(* Logix 5000 project; controller cal1615 1756-L62 rev 20.19; software revision 20.05; part 8 of 82 *)
(* tags used below, declared in another part *)
   AFI : BOOL;   // Always False Bit
   AutoT : PIDE_AUTOTUNE;
   FAULT : BOOL;   // Fault AFI
   HMI : BOOL;   // AFI HMI
   p01_dint_to_hmi : DINT[16];   // System Dint to HMI
   p01_param_heater_hl : REAL;   // Machine Parameter Heater HighTemperature Max Limit
   p01_param_process_air_hl : REAL;   // Machine Parameter Process Air High Limit
   p01_param_process_air_max : REAL;   // Machine Parameter Process Air High Temperature Max Setpoint Limit
   p01_param_temp_limit : REAL;   // Machine Parameter Maximum Temperature for Fan Operation
   p01_recipe_active : recipe;   // Active Recipe
   p01r01 : routine;
   p01r02 : routine;   // System Misc Control
   p01r02_all_fans_stopped : BOOL;   // System Misc Control All Fans Stopped
   p01r02_batch_run_time : DINT;   // System Misc Control Batch Minutes
   p01r02_batch_run_time_hrs : DINT;   // System Misc Control Batch Hours
   p01r02_ethernet_comm : DINT;
   p01r02_fault_exists : BOOL;
   p01r02_flash_bit : BOOL;   // System Misc Control Flash Bit
   p01r02_flash_timer_off : TIMER;   // System Misc Control Flash Timer Off
   p01r02_flash_timer_on : TIMER;   // System Misc Control Flash Timer On
   p01r02_plc_faults : DINT;   // System Misc Control PLC Faults
   p01r02_plc_scan_time : DINT;   // System PLC Scan Time
   p01r02_plc_scan_time_in_sec : REAL;   // System PLC Scan Time in Seconds
   p01r02_timer_batch : TIMER;   // System Misc Control Batch Timer Seconds
   p01r02_timer_fault : TIMER[25];   // System Misc Control Fault Dwell Timer
   p01r02_timer_half_second_off : TIMER;   // System Misc Control Timer Second Pulse Off
   p01r02_timer_half_second_on : TIMER;   // System Misc Control Timer 1/2 Second Pulse On
   p01r02_timer_second : TIMER[2];   // System Misc Control Timer Second Pulse
   p01r02_unack_fault : BOOL;   // System Misc Control Unacknowledged Fault Exists
   p01r02_unack_warning : BOOL;   // System Misc Control Unacknowledged Warning Exists
   p01r02_vfd_comm_2 : DINT[50];
   p01r02_warnings_exists : BOOL;
   p01r03 : routine;   // System Inputs
   p01r04 : routine;   // System Outputs
   p01r05 : routine;   // System Dint to HMI
   p01r06 : routine;   // System Real to HMI
   p01r07 : routine;   // System Alarms
   p01r08 : routine;   // System Warnings
   p01r09 : routine;   // System Modes
   p01r09_pb_global_reset : BOOL;   // System Modes PB: Global Fault Reset
   p01r10 : routine;   // System Annunciators
   p01r11 : routine;   // System Timer Presets
   p01r12 : routine;   // System Line Accel Decel Control
   p01r13 : routine;   // System Line Start Sequence
   p01r13_line_running : BOOL;   // System Line Start Sequence Line Running
   p02_dint_from_hmi : hmi_dint;
   p11r31_request_auto_run : BOOL;   // Zone 1 Exhaust Fan Run Request
   p11r32_request_auto_run : BOOL;   // Zone 1 Recirc Fan Run Request
   p12r31_request_auto_run : BOOL;   // Zone 2 Exhaust Fan Run Request
   p12r32_request_auto_run : BOOL;   // Zone 2 Recirc Fan Run Request
   p13r31_request_auto_run : BOOL;   // Zone 3 Exhaust Fan Run Request
   p13r32_request_auto_run : BOOL;   // Zone 3 Recirc Fan Run Request
   p23_do_enable_impreg_exhaust_fan : BOOL;   // Impreg Enclosure Digital Output Exhaust Fan Enable
   p23r13_request_auto_run : BOOL;   // Impreg Supply Fan VFD Request Auto Run
   p25_ai_ts2_lc : REAL;   // System Metering Roll VFD Minimum Start Tension
   p25r10_pid_manual_request : BOOL;
   p25r10_tension_request : BOOL;
   p25r20_pide_cv : REAL;

        [421] := 3.25, [422] := 3.25, [423] := 3.25, [424] := 3.25, [425] := 3.25, [426] := 3.25, [427] := 3.25, [428] := 3.25, [429] := 3.25, [430] := 3.25, [431] := 3.25, [432] := 3.25, [433] := 3.25, [434] := 3.25, [435] := 3.25, [436] := 3.25, [437] := 3.25, [438] := 3.25, [439] := 3.25, [440] := 3.25, [441] := 3.25, [442] := 3.25, [443] := 3.25, [444] := 3.25, [445] := 3.25, [446] := 3.25, [447] := 3.25, [448] := 3.25, [449] := 3.25, [450] := 3.25, [451] := 3.25, [452] := 3.25, [453] := 3.25, [454] := 3.25, [455] := 3.25, [456] := 3.25, [457] := 3.25, [458] := 3.25, [459] := 3.25, [460] := 3.25, [461] := 3.25, [462] := 3.25, [463] := 3.25, [464] := 3.25, [465] := 3.25, [466] := 3.25, [467] := 3.25, [468] := 3.25, [469] := 3.25, [470] := 3.25, [471] := 3.25, [472] := 3.25, [473] := 3.25, [474] := 3.25, [475] := 3.25, [476] := 3.25, [477] := 3.25, [478] := 3.25, [479] := 3.25, [480] := 3.25,
        [481] := 3.25, [482] := 3.25, [483] := 3.25, [484] := 3.25, [485] := 3.25, [486] := 3.25, [487] := 3.25, [488] := 3.25, [489] := 3.25, [490] := 3.25, [491] := 3.25, [492] := 3.25, [493] := 3.25, [494] := 3.25, [495] := 3.25, [496] := 3.25, [497] := 3.25, [498] := 3.25, [499] := 3.25, [500] := 3.25, [501] := 3.25, [502] := 3.25, [503] := 3.25, [504] := 3.25, [505] := 3.25, [506] := 3.25, [507] := 3.25, [508] := 3.25, [509] := 3.25, [510] := 3.25, [511] := 3.25, [512] := 3.25, [513] := 3.25, [514] := 3.25, [515] := 3.25, [516] := 3.25, [517] := 3.25, [518] := 3.25, [519] := 3.25, [520] := 3.25, [521] := 3.25, [522] := 3.25, [523] := 3.25, [524] := 3.25, [525] := 3.25, [526] := 3.25, [527] := 3.25, [528] := 3.25, [529] := 3.25, [530] := 3.25, [531] := 3.25, [532] := 3.25, [533] := 3.25, [534] := 3.25, [535] := 3.25, [536] := 3.25, [537] := 3.25, [538] := 3.25, [539] := 3.25, [540] := 3.25,
        [541] := 3.25, [542] := 3.25, [543] := 3.25, [544] := 3.25, [545] := 3.25, [546] := 3.25, [547] := 3.25, [548] := 3.25, [549] := 3.25, [550] := 3.25, [551] := 3.25, [552] := 3.25, [553] := 3.25, [554] := 3.25, [555] := 3.25, [556] := 3.25, [557] := 3.25, [558] := 3.25, [559] := 3.25, [560] := 3.25, [561] := 3.25, [562] := 3.25, [563] := 3.25, [564] := 3.25, [565] := 3.25, [566] := 3.25, [567] := 3.25, [568] := 3.25, [569] := 3.25, [570] := 3.25, [571] := 3.25, [572] := 3.25, [573] := 3.25, [574] := 3.25, [575] := 3.25, [576] := 3.25, [577] := 3.25, [578] := 3.25, [579] := 3.25, [580] := 3.25, [581] := 3.25, [582] := 3.25, [583] := 3.25, [584] := 3.25, [585] := 3.25, [586] := 3.25, [587] := 3.25, [588] := 3.25, [589] := 3.25, [590] := 3.25, [591] := 3.25, [592] := 3.25, [593] := 3.25, [594] := 3.25, [595] := 3.25, [596] := 3.25, [597] := 3.25, [598] := 3.25, [599] := 3.25, [600] := 3.25,
        [601] := 3.25, [602] := 3.25, [603] := 3.25, [604] := 3.25, [605] := 3.25, [606] := 3.25, [607] := 3.25, [608] := 3.25, [609] := 3.25, [610] := 3.25, [611] := 3.25, [612] := 3.25, [613] := 3.25, [614] := 3.25, [615] := 3.25, [616] := 3.25, [617] := 3.25, [618] := 3.25, [619] := 3.25, [620] := 3.25, [621] := 3.25, [622] := 3.25, [623] := 3.25, [624] := 3.25, [625] := 3.25, [626] := 3.25, [627] := 3.25, [628] := 3.25, [629] := 3.25, [630] := 3.25, [631] := 3.25, [632] := 3.25, [633] := 3.25, [634] := 3.25, [635] := 3.25, [636] := 3.25, [637] := 3.25, [638] := 3.25, [639] := 3.25, [640] := 3.25, [641] := 3.25, [642] := 3.25, [643] := 3.25, [644] := 3.25, [645] := 3.25, [646] := 3.25, [647] := 3.25, [648] := 3.25, [649] := 3.25, [650] := 3.25, [651] := 3.25, [652] := 3.25, [653] := 3.25, [654] := 3.25, [655] := 3.25, [656] := 3.25, [657] := 3.25, [658] := 3.25, [659] := 3.25, [660] := 3.25,
        [661] := 3.25, [662] := 3.25, [663] := 3.25, [664] := 3.25, [665] := 3.25, [666] := 3.25, [667] := 3.25, [668] := 3.25, [669] := 3.25, [670] := 3.25, [671] := 3.25, [672] := 3.25, [673] := 3.25, [674] := 3.25, [675] := 3.25, [676] := 3.25, [677] := 3.25, [678] := 3.25, [679] := 3.25, [680] := 3.25, [681] := 3.25, [682] := 3.25, [683] := 3.25, [684] := 3.25, [685] := 3.25, [686] := 3.25, [687] := 3.25, [688] := 3.25, [689] := 3.25, [690] := 3.25, [691] := 3.25, [692] := 3.25, [693] := 3.25, [694] := 3.25, [695] := 3.25, [696] := 3.25, [697] := 3.25, [698] := 3.25, [699] := 3.25, [700] := 3.25, [701] := 3.25, [702] := 3.25, [703] := 3.25, [704] := 3.25, [705] := 3.25, [706] := 3.25, [707] := 3.25, [708] := 3.25, [709] := 3.25, [710] := 3.25, [711] := 3.25, [712] := 3.25, [713] := 3.25, [714] := 3.25, [715] := 3.25, [716] := 3.25, [717] := 3.25, [718] := 3.25, [719] := 3.25, [720] := 3.25,
        [721] := 3.25, [722] := 3.25, [723] := 3.25, [724] := 3.25, [725] := 3.25, [726] := 3.25, [727] := 3.25, [728] := 3.25, [729] := 3.25, [730] := 3.25, [731] := 3.25, [732] := 3.25, [733] := 3.25, [734] := 3.25, [735] := 3.25, [736] := 3.25, [737] := 3.25, [738] := 3.25, [739] := 3.25, [740] := 3.25, [741] := 3.25, [742] := 3.25, [743] := 3.25, [744] := 3.25, [745] := 3.25, [746] := 3.25, [747] := 3.25, [748] := 3.25, [749] := 3.25, [750] := 3.25, [751] := 3.25, [752] := 3.25, [753] := 3.25, [754] := 3.25, [755] := 3.25, [756] := 3.25, [757] := 3.25, [758] := 3.25, [759] := 3.25, [760] := 3.25, [761] := 3.25, [762] := 3.25, [763] := 3.25, [764] := 3.25, [765] := 3.25, [766] := 3.25, [767] := 3.25, [768] := 3.25, [769] := 3.25, [770] := 3.25, [771] := 3.25, [772] := 3.25, [773] := 3.25, [774] := 3.25, [775] := 3.25, [776] := 3.25, [777] := 3.25, [778] := 3.25, [779] := 3.25, [780] := 3.25,
        [781] := 3.25, [782] := 3.25, [783] := 3.25, [784] := 3.25, [785] := 3.25, [786] := 3.25, [787] := 3.25, [788] := 3.25, [789] := 3.25, [790] := 3.25, [791] := 3.25, [792] := 3.25, [793] := 3.25, [794] := 3.25, [795] := 3.25, [796] := 3.25, [797] := 3.25, [798] := 3.25, [799] := 3.25, [800] := 3.25, [801] := 3.25, [802] := 3.25, [803] := 3.25, [804] := 3.25, [805] := 3.25, [806] := 3.25, [807] := 3.25, [808] := 3.25, [809] := 3.25, [810] := 3.25, [811] := 3.25, [812] := 3.25, [813] := 3.25, [814] := 3.25, [815] := 3.25, [816] := 3.25, [817] := 3.25, [818] := 3.25, [819] := 3.25, [820] := 3.25, [821] := 3.25, [822] := 3.25, [823] := 3.25, [824] := 3.25, [825] := 3.25, [826] := 3.25, [827] := 3.25, [828] := 3.25, [829] := 3.25, [830] := 3.25, [831] := 3.25, [832] := 3.25, [833] := 3.25, [834] := 3.25, [835] := 3.25, [836] := 3.25, [837] := 3.25, [838] := 3.25, [839] := 3.25, [840] := 3.25,
        [841] := 3.25, [842] := 3.25, [843] := 3.25, [844] := 3.25, [845] := 3.25, [846] := 3.25, [847] := 3.25, [848] := 3.25, [849] := 3.25, [850] := 3.25, [851] := 3.25, [852] := 3.25, [853] := 3.25, [854] := 3.25, [855] := 3.25, [856] := 3.25, [857] := 3.25, [858] := 3.25, [859] := 3.25, [860] := 3.25, [861] := 3.25, [862] := 3.25, [863] := 3.25, [864] := 3.25, [865] := 3.25, [866] := 3.25, [867] := 3.25, [868] := 3.25, [869] := 3.25, [870] := 3.25, [871] := 3.25, [872] := 3.25, [873] := 3.25, [874] := 3.25, [875] := 3.25, [876] := 3.25, [877] := 3.25, [878] := 3.25, [879] := 3.25, [880] := 3.25, [881] := 3.25, [882] := 3.25, [883] := 3.25, [884] := 3.25, [885] := 3.25, [886] := 3.25, [887] := 3.25, [888] := 3.25, [889] := 3.25, [890] := 3.25, [891] := 3.25, [892] := 3.25, [893] := 3.25, [894] := 3.25, [895] := 3.25, [896] := 3.25, [897] := 3.25, [898] := 3.25, [899] := 3.25, [900] := 3.25,
        [901] := 3.25, [902] := 3.25, [903] := 3.25, [904] := 3.25, [905] := 3.25, [906] := 3.25, [907] := 3.25, [908] := 3.25, [909] := 3.25, [910] := 3.25, [911] := 3.25, [912] := 3.25, [913] := 3.25, [914] := 3.25, [915] := 3.25, [916] := 3.25, [917] := 3.25, [918] := 3.25, [919] := 3.25, [920] := 3.25, [921] := 3.25, [922] := 3.25, [923] := 3.25, [924] := 3.25, [925] := 3.25, [926] := 3.25, [927] := 3.25, [928] := 3.25, [929] := 3.25, [930] := 3.25, [931] := 3.25, [932] := 3.25, [933] := 3.25, [934] := 3.25, [935] := 3.25, [936] := 3.25, [937] := 3.25, [938] := 3.25, [939] := 3.25, [940] := 3.25, [941] := 3.25, [942] := 3.25, [943] := 3.25, [944] := 3.25, [945] := 3.25, [946] := 3.25, [947] := 3.25, [948] := 3.25, [949] := 3.25, [950] := 3.25, [951] := 3.25, [952] := 3.25, [953] := 3.25, [954] := 3.25, [955] := 3.25, [956] := 3.25, [957] := 3.25, [958] := 3.25, [959] := 3.25, [960] := 3.25,
        [961] := 3.25, [962] := 3.25, [963] := 3.25, [964] := 3.25, [965] := 3.25, [966] := 3.25, [967] := 3.25, [968] := 3.25, [969] := 3.25, [970] := 3.25, [971] := 3.25, [972] := 3.25, [973] := 3.25, [974] := 3.25, [975] := 3.25, [976] := 3.25, [977] := 3.25, [978] := 3.25, [979] := 3.25, [980] := 3.25, [981] := 3.25, [982] := 3.25, [983] := 3.25, [984] := 3.25, [985] := 3.25, [986] := 3.25, [987] := 3.25, [988] := 3.25, [989] := 3.25, [990] := 3.25, [991] := 3.25, [992] := 3.25, [993] := 3.25, [994] := 3.25, [995] := 3.25, [996] := 3.25, [997] := 3.25, [998] := 3.25, [999] := 3.25);
   p29r17_winder_a_selected_diam_inch : REAL := 3.25;   // Winder Winder A Diameter Calculation Winder Selected Diameter [in]
   p29r17_winder_a_unload : REAL := 4.77611;
   p29r18 : routine := (comment := -1073741777);   // Winder Winder B Diameter
        .UNACK_FAULT   // Winder Winder B Diameter Unacknowleged Faults Exist
        .UNACK_WARNING   // Winder Winder B Diameter Unacknowleged Warnings Exist
   p29r18_ave_control : CONTROL := (LEN := 19);   // Winder Winder A Diameter Calculation AVE Control
   p29r18_diameter_calc_active : BOOL;   // Winder Winder B Diameter Calculation Calculation Active
   p29r18_min_tension : REAL := 10.0;   // Winder Winder B Diameter Calc Minimum Tension
   p29r18_selected_core_diameter : REAL := 6.0;   // Winder Winder B Diameter Calculation Selected Core Diameter
   p29r18_stack_ctrl : CONTROL := (LEN := 20, POS := 19);   // Winder Winder B Diameter Calculation FiFo Control
   p29r18_timer : TIMER[5] := ([0].PRE := 20000, [1].PRE := 500);   // Winder Winder B Diameter Calculation Timers
   p29r18_timer_fault : TIMER[4];   // Winder Winder B Diameter Calculation Fault Dwell Timer
   p29r18_timer_warning : TIMER[4];   // Winder Winder B Diameter Warning Dwell Timer
   p29r18_winder_b_actual_diam_inch : REAL := 6.0;   // Winder Winder B Diameter Calculation Actual Diameter [in]
   p29r18_winder_b_avg_diam_inch : REAL := 6.0;   // Winder Winder B Diameter Calculation Average Diameter [in]
   p29r18_winder_b_calc_diam_inch : REAL := 6.0;   // Winder Winder B Diameter Calculated Diameter Inch
   p29r18_winder_b_diam_avg_stack : REAL[1000] := ([0] := 6.0, [1] := 6.0, [2] := 6.0, [3] := 6.0, [4] := 6.0, [5] := 6.0, [6] := 6.0, [7] := 6.0, [8] := 6.0, [9] := 6.0, [10] := 6.0, [11] := 6.0, [12] := 6.0, [13] := 6.0, [14] := 6.0, [15] := 6.0, [16] := 6.0, [17] := 6.0, [18] := 6.0, [19] := 6.0, [20] := 6.0, [21] := 6.0, [22] := 6.0, [23] := 6.0, [24] := 6.0, [25] := 6.0, [26] := 6.0, [27] := 6.0, [28] := 6.0, [29] := 6.0, [30] := 6.0, [31] := 6.0, [32] := 6.0, [33] := 6.0, [34] := 6.0, [35] := 6.0, [36] := 6.0, [37] := 6.0, [38] := 6.0, [39] := 6.0, [40] := 6.0, [41] := 6.0, [42] := 6.0, [43] := 6.0, [44] := 6.0, [45] := 6.0, [46] := 6.0, [47] := 6.0, [48] := 6.0, [49] := 6.0, [50] := 6.0, [51] := 6.0, [52] := 6.0, [53] := 6.0, [54] := 6.0, [55] := 6.0, [56] := 6.0, [57] := 6.0, [58] := 6.0, [59] := 6.0,
        [60] := 6.0, [61] := 6.0, [62] := 6.0, [63] := 6.0, [64] := 6.0, [65] := 6.0, [66] := 6.0, [67] := 6.0, [68] := 6.0, [69] := 6.0, [70] := 6.0, [71] := 6.0, [72] := 6.0, [73] := 6.0, [74] := 6.0, [75] := 6.0, [76] := 6.0, [77] := 6.0, [78] := 6.0, [79] := 6.0, [80] := 6.0, [81] := 6.0, [82] := 6.0, [83] := 6.0, [84] := 6.0, [85] := 6.0, [86] := 6.0, [87] := 6.0, [88] := 6.0, [89] := 6.0, [90] := 6.0, [91] := 6.0, [92] := 6.0, [93] := 6.0, [94] := 6.0, [95] := 6.0, [96] := 6.0, [97] := 6.0, [98] := 6.0, [99] := 6.0, [100] := 6.0, [101] := 6.0, [102] := 6.0, [103] := 6.0, [104] := 6.0, [105] := 6.0, [106] := 6.0, [107] := 6.0, [108] := 6.0, [109] := 6.0, [110] := 6.0, [111] := 6.0, [112] := 6.0, [113] := 6.0, [114] := 6.0, [115] := 6.0, [116] := 6.0, [117] := 6.0, [118] := 6.0, [119] := 6.0,
        [120] := 6.0, [121] := 6.0, [122] := 6.0, [123] := 6.0, [124] := 6.0, [125] := 6.0, [126] := 6.0, [127] := 6.0, [128] := 6.0, [129] := 6.0, [130] := 6.0, [131] := 6.0, [132] := 6.0, [133] := 6.0, [134] := 6.0, [135] := 6.0, [136] := 6.0, [137] := 6.0, [138] := 6.0, [139] := 6.0, [140] := 6.0, [141] := 6.0, [142] := 6.0, [143] := 6.0, [144] := 6.0, [145] := 6.0, [146] := 6.0, [147] := 6.0, [148] := 6.0, [149] := 6.0, [150] := 6.0, [151] := 6.0, [152] := 6.0, [153] := 6.0, [154] := 6.0, [155] := 6.0, [156] := 6.0, [157] := 6.0, [158] := 6.0, [159] := 6.0, [160] := 6.0, [161] := 6.0, [162] := 6.0, [163] := 6.0, [164] := 6.0, [165] := 6.0, [166] := 6.0, [167] := 6.0, [168] := 6.0, [169] := 6.0, [170] := 6.0, [171] := 6.0, [172] := 6.0, [173] := 6.0, [174] := 6.0, [175] := 6.0, [176] := 6.0, [177] := 6.0, [178] := 6.0, [179] := 6.0,
        [180] := 6.0, [181] := 6.0, [182] := 6.0, [183] := 6.0, [184] := 6.0, [185] := 6.0, [186] := 6.0, [187] := 6.0, [188] := 6.0, [189] := 6.0, [190] := 6.0, [191] := 6.0, [192] := 6.0, [193] := 6.0, [194] := 6.0, [195] := 6.0, [196] := 6.0, [197] := 6.0, [198] := 6.0, [199] := 6.0, [200] := 6.0, [201] := 6.0, [202] := 6.0, [203] := 6.0, [204] := 6.0, [205] := 6.0, [206] := 6.0, [207] := 6.0, [208] := 6.0, [209] := 6.0, [210] := 6.0, [211] := 6.0, [212] := 6.0, [213] := 6.0, [214] := 6.0, [215] := 6.0, [216] := 6.0, [217] := 6.0, [218] := 6.0, [219] := 6.0, [220] := 6.0, [221] := 6.0, [222] := 6.0, [223] := 6.0, [224] := 6.0, [225] := 6.0, [226] := 6.0, [227] := 6.0, [228] := 6.0, [229] := 6.0, [230] := 6.0, [231] := 6.0, [232] := 6.0, [233] := 6.0, [234] := 6.0, [235] := 6.0, [236] := 6.0, [237] := 6.0, [238] := 6.0, [239] := 6.0,
        [240] := 6.0, [241] := 6.0, [242] := 6.0, [243] := 6.0, [244] := 6.0, [245] := 6.0, [246] := 6.0, [247] := 6.0, [248] := 6.0, [249] := 6.0, [250] := 6.0, [251] := 6.0, [252] := 6.0, [253] := 6.0, [254] := 6.0, [255] := 6.0, [256] := 6.0, [257] := 6.0, [258] := 6.0, [259] := 6.0, [260] := 6.0, [261] := 6.0, [262] := 6.0, [263] := 6.0, [264] := 6.0, [265] := 6.0, [266] := 6.0, [267] := 6.0, [268] := 6.0, [269] := 6.0, [270] := 6.0, [271] := 6.0, [272] := 6.0, [273] := 6.0, [274] := 6.0, [275] := 6.0, [276] := 6.0, [277] := 6.0, [278] := 6.0, [279] := 6.0, [280] := 6.0, [281] := 6.0, [282] := 6.0, [283] := 6.0, [284] := 6.0, [285] := 6.0, [286] := 6.0, [287] := 6.0, [288] := 6.0, [289] := 6.0, [290] := 6.0, [291] := 6.0, [292] := 6.0, [293] := 6.0, [294] := 6.0, [295] := 6.0, [296] := 6.0, [297] := 6.0, [298] := 6.0, [299] := 6.0,
        [300] := 6.0, [301] := 6.0, [302] := 6.0, [303] := 6.0, [304] := 6.0, [305] := 6.0, [306] := 6.0, [307] := 6.0, [308] := 6.0, [309] := 6.0, [310] := 6.0, [311] := 6.0, [312] := 6.0, [313] := 6.0, [314] := 6.0, [315] := 6.0, [316] := 6.0, [317] := 6.0, [318] := 6.0, [319] := 6.0, [320] := 6.0, [321] := 6.0, [322] := 6.0, [323] := 6.0, [324] := 6.0, [325] := 6.0, [326] := 6.0, [327] := 6.0, [328] := 6.0, [329] := 6.0, [330] := 6.0, [331] := 6.0, [332] := 6.0, [333] := 6.0, [334] := 6.0, [335] := 6.0, [336] := 6.0, [337] := 6.0, [338] := 6.0, [339] := 6.0, [340] := 6.0, [341] := 6.0, [342] := 6.0, [343] := 6.0, [344] := 6.0, [345] := 6.0, [346] := 6.0, [347] := 6.0, [348] := 6.0, [349] := 6.0, [350] := 6.0, [351] := 6.0, [352] := 6.0, [353] := 6.0, [354] := 6.0, [355] := 6.0, [356] := 6.0, [357] := 6.0, [358] := 6.0, [359] := 6.0,
        [360] := 6.0, [361] := 6.0, [362] := 6.0, [363] := 6.0, [364] := 6.0, [365] := 6.0, [366] := 6.0, [367] := 6.0, [368] := 6.0, [369] := 6.0, [370] := 6.0, [371] := 6.0, [372] := 6.0, [373] := 6.0, [374] := 6.0, [375] := 6.0, [376] := 6.0, [377] := 6.0, [378] := 6.0, [379] := 6.0, [380] := 6.0, [381] := 6.0, [382] := 6.0, [383] := 6.0, [384] := 6.0, [385] := 6.0, [386] := 6.0, [387] := 6.0, [388] := 6.0, [389] := 6.0, [390] := 6.0, [391] := 6.0, [392] := 6.0, [393] := 6.0, [394] := 6.0, [395] := 6.0, [396] := 6.0, [397] := 6.0, [398] := 6.0, [399] := 6.0, [400] := 6.0, [401] := 6.0, [402] := 6.0, [403] := 6.0, [404] := 6.0, [405] := 6.0, [406] := 6.0, [407] := 6.0, [408] := 6.0, [409] := 6.0, [410] := 6.0, [411] := 6.0, [412] := 6.0, [413] := 6.0, [414] := 6.0, [415] := 6.0, [416] := 6.0, [417] := 6.0, [418] := 6.0, [419] := 6.0,
        [420] := 6.0, [421] := 6.0, [422] := 6.0, [423] := 6.0, [424] := 6.0, [425] := 6.0, [426] := 6.0, [427] := 6.0, [428] := 6.0, [429] := 6.0, [430] := 6.0, [431] := 6.0, [432] := 6.0, [433] := 6.0, [434] := 6.0, [435] := 6.0, [436] := 6.0, [437] := 6.0, [438] := 6.0, [439] := 6.0, [440] := 6.0, [441] := 6.0, [442] := 6.0, [443] := 6.0, [444] := 6.0, [445] := 6.0, [446] := 6.0, [447] := 6.0, [448] := 6.0, [449] := 6.0, [450] := 6.0, [451] := 6.0, [452] := 6.0, [453] := 6.0, [454] := 6.0, [455] := 6.0, [456] := 6.0, [457] := 6.0, [458] := 6.0, [459] := 6.0, [460] := 6.0, [461] := 6.0, [462] := 6.0, [463] := 6.0, [464] := 6.0, [465] := 6.0, [466] := 6.0, [467] := 6.0, [468] := 6.0, [469] := 6.0, [470] := 6.0, [471] := 6.0, [472] := 6.0, [473] := 6.0, [474] := 6.0, [475] := 6.0, [476] := 6.0, [477] := 6.0, [478] := 6.0, [479] := 6.0,
        [480] := 6.0, [481] := 6.0, [482] := 6.0, [483] := 6.0, [484] := 6.0, [485] := 6.0, [486] := 6.0, [487] := 6.0, [488] := 6.0, [489] := 6.0, [490] := 6.0, [491] := 6.0, [492] := 6.0, [493] := 6.0, [494] := 6.0, [495] := 6.0, [496] := 6.0, [497] := 6.0, [498] := 6.0, [499] := 6.0, [500] := 6.0, [501] := 6.0, [502] := 6.0, [503] := 6.0, [504] := 6.0, [505] := 6.0, [506] := 6.0, [507] := 6.0, [508] := 6.0, [509] := 6.0, [510] := 6.0, [511] := 6.0, [512] := 6.0, [513] := 6.0, [514] := 6.0, [515] := 6.0, [516] := 6.0, [517] := 6.0, [518] := 6.0, [519] := 6.0, [520] := 6.0, [521] := 6.0, [522] := 6.0, [523] := 6.0, [524] := 6.0, [525] := 6.0, [526] := 6.0, [527] := 6.0, [528] := 6.0, [529] := 6.0, [530] := 6.0, [531] := 6.0, [532] := 6.0, [533] := 6.0, [534] := 6.0, [535] := 6.0, [536] := 6.0, [537] := 6.0, [538] := 6.0, [539] := 6.0,
        [540] := 6.0, [541] := 6.0, [542] := 6.0, [543] := 6.0, [544] := 6.0, [545] := 6.0, [546] := 6.0, [547] := 6.0, [548] := 6.0, [549] := 6.0, [550] := 6.0, [551] := 6.0, [552] := 6.0, [553] := 6.0, [554] := 6.0, [555] := 6.0, [556] := 6.0, [557] := 6.0, [558] := 6.0, [559] := 6.0, [560] := 6.0, [561] := 6.0, [562] := 6.0, [563] := 6.0, [564] := 6.0, [565] := 6.0, [566] := 6.0, [567] := 6.0, [568] := 6.0, [569] := 6.0, [570] := 6.0, [571] := 6.0, [572] := 6.0, [573] := 6.0, [574] := 6.0, [575] := 6.0, [576] := 6.0, [577] := 6.0, [578] := 6.0, [579] := 6.0, [580] := 6.0, [581] := 6.0, [582] := 6.0, [583] := 6.0, [584] := 6.0, [585] := 6.0, [586] := 6.0, [587] := 6.0, [588] := 6.0, [589] := 6.0, [590] := 6.0, [591] := 6.0, [592] := 6.0, [593] := 6.0, [594] := 6.0, [595] := 6.0, [596] := 6.0, [597] := 6.0, [598] := 6.0, [599] := 6.0,
        [600] := 6.0, [601] := 6.0, [602] := 6.0, [603] := 6.0, [604] := 6.0, [605] := 6.0, [606] := 6.0, [607] := 6.0, [608] := 6.0, [609] := 6.0, [610] := 6.0, [611] := 6.0, [612] := 6.0, [613] := 6.0, [614] := 6.0, [615] := 6.0, [616] := 6.0, [617] := 6.0, [618] := 6.0, [619] := 6.0, [620] := 6.0, [621] := 6.0, [622] := 6.0, [623] := 6.0, [624] := 6.0, [625] := 6.0, [626] := 6.0, [627] := 6.0, [628] := 6.0, [629] := 6.0, [630] := 6.0, [631] := 6.0, [632] := 6.0, [633] := 6.0, [634] := 6.0, [635] := 6.0, [636] := 6.0, [637] := 6.0, [638] := 6.0, [639] := 6.0, [640] := 6.0, [641] := 6.0, [642] := 6.0, [643] := 6.0, [644] := 6.0, [645] := 6.0, [646] := 6.0, [647] := 6.0, [648] := 6.0, [649] := 6.0, [650] := 6.0, [651] := 6.0, [652] := 6.0, [653] := 6.0, [654] := 6.0, [655] := 6.0, [656] := 6.0, [657] := 6.0, [658] := 6.0, [659] := 6.0,
        [660] := 6.0, [661] := 6.0, [662] := 6.0, [663] := 6.0, [664] := 6.0, [665] := 6.0, [666] := 6.0, [667] := 6.0, [668] := 6.0, [669] := 6.0, [670] := 6.0, [671] := 6.0, [672] := 6.0, [673] := 6.0, [674] := 6.0, [675] := 6.0, [676] := 6.0, [677] := 6.0, [678] := 6.0, [679] := 6.0, [680] := 6.0, [681] := 6.0, [682] := 6.0, [683] := 6.0, [684] := 6.0, [685] := 6.0, [686] := 6.0, [687] := 6.0, [688] := 6.0, [689] := 6.0, [690] := 6.0, [691] := 6.0, [692] := 6.0, [693] := 6.0, [694] := 6.0, [695] := 6.0, [696] := 6.0, [697] := 6.0, [698] := 6.0, [699] := 6.0, [700] := 6.0, [701] := 6.0, [702] := 6.0, [703] := 6.0, [704] := 6.0, [705] := 6.0, [706] := 6.0, [707] := 6.0, [708] := 6.0, [709] := 6.0, [710] := 6.0, [711] := 6.0, [712] := 6.0, [713] := 6.0, [714] := 6.0, [715] := 6.0, [716] := 6.0, [717] := 6.0, [718] := 6.0, [719] := 6.0,
        [720] := 6.0, [721] := 6.0, [722] := 6.0, [723] := 6.0, [724] := 6.0, [725] := 6.0, [726] := 6.0, [727] := 6.0, [728] := 6.0, [729] := 6.0, [730] := 6.0, [731] := 6.0, [732] := 6.0, [733] := 6.0, [734] := 6.0, [735] := 6.0, [736] := 6.0, [737] := 6.0, [738] := 6.0, [739] := 6.0, [740] := 6.0, [741] := 6.0, [742] := 6.0, [743] := 6.0, [744] := 6.0, [745] := 6.0, [746] := 6.0, [747] := 6.0, [748] := 6.0, [749] := 6.0, [750] := 6.0, [751] := 6.0, [752] := 6.0, [753] := 6.0, [754] := 6.0, [755] := 6.0, [756] := 6.0, [757] := 6.0, [758] := 6.0, [759] := 6.0, [760] := 6.0, [761] := 6.0, [762] := 6.0, [763] := 6.0, [764] := 6.0, [765] := 6.0, [766] := 6.0, [767] := 6.0, [768] := 6.0, [769] := 6.0, [770] := 6.0, [771] := 6.0, [772] := 6.0, [773] := 6.0, [774] := 6.0, [775] := 6.0, [776] := 6.0, [777] := 6.0, [778] := 6.0, [779] := 6.0,
        [780] := 6.0, [781] := 6.0, [782] := 6.0, [783] := 6.0, [784] := 6.0, [785] := 6.0, [786] := 6.0, [787] := 6.0, [788] := 6.0, [789] := 6.0, [790] := 6.0, [791] := 6.0, [792] := 6.0, [793] := 6.0, [794] := 6.0, [795] := 6.0, [796] := 6.0, [797] := 6.0, [798] := 6.0, [799] := 6.0, [800] := 6.0, [801] := 6.0, [802] := 6.0, [803] := 6.0, [804] := 6.0, [805] := 6.0, [806] := 6.0, [807] := 6.0, [808] := 6.0, [809] := 6.0, [810] := 6.0, [811] := 6.0, [812] := 6.0, [813] := 6.0, [814] := 6.0, [815] := 6.0, [816] := 6.0, [817] := 6.0, [818] := 6.0, [819] := 6.0, [820] := 6.0, [821] := 6.0, [822] := 6.0, [823] := 6.0, [824] := 6.0, [825] := 6.0, [826] := 6.0, [827] := 6.0, [828] := 6.0, [829] := 6.0, [830] := 6.0, [831] := 6.0, [832] := 6.0, [833] := 6.0, [834] := 6.0, [835] := 6.0, [836] := 6.0, [837] := 6.0, [838] := 6.0, [839] := 6.0,
        [840] := 6.0, [841] := 6.0, [842] := 6.0, [843] := 6.0, [844] := 6.0, [845] := 6.0, [846] := 6.0, [847] := 6.0, [848] := 6.0, [849] := 6.0, [850] := 6.0, [851] := 6.0, [852] := 6.0, [853] := 6.0, [854] := 6.0, [855] := 6.0, [856] := 6.0, [857] := 6.0, [858] := 6.0, [859] := 6.0, [860] := 6.0, [861] := 6.0, [862] := 6.0, [863] := 6.0, [864] := 6.0, [865] := 6.0, [866] := 6.0, [867] := 6.0, [868] := 6.0, [869] := 6.0, [870] := 6.0, [871] := 6.0, [872] := 6.0, [873] := 6.0, [874] := 6.0, [875] := 6.0, [876] := 6.0, [877] := 6.0, [878] := 6.0, [879] := 6.0, [880] := 6.0, [881] := 6.0, [882] := 6.0, [883] := 6.0, [884] := 6.0, [885] := 6.0, [886] := 6.0, [887] := 6.0, [888] := 6.0, [889] := 6.0, [890] := 6.0, [891] := 6.0, [892] := 6.0, [893] := 6.0, [894] := 6.0, [895] := 6.0, [896] := 6.0, [897] := 6.0, [898] := 6.0, [899] := 6.0,
        [900] := 6.0, [901] := 6.0, [902] := 6.0, [903] := 6.0, [904] := 6.0, [905] := 6.0, [906] := 6.0, [907] := 6.0, [908] := 6.0, [909] := 6.0, [910] := 6.0, [911] := 6.0, [912] := 6.0, [913] := 6.0, [914] := 6.0, [915] := 6.0, [916] := 6.0, [917] := 6.0, [918] := 6.0, [919] := 6.0, [920] := 6.0, [921] := 6.0, [922] := 6.0, [923] := 6.0, [924] := 6.0, [925] := 6.0, [926] := 6.0, [927] := 6.0, [928] := 6.0, [929] := 6.0, [930] := 6.0, [931] := 6.0, [932] := 6.0, [933] := 6.0, [934] := 6.0, [935] := 6.0, [936] := 6.0, [937] := 6.0, [938] := 6.0, [939] := 6.0, [940] := 6.0, [941] := 6.0, [942] := 6.0, [943] := 6.0, [944] := 6.0, [945] := 6.0, [946] := 6.0, [947] := 6.0, [948] := 6.0, [949] := 6.0, [950] := 6.0, [951] := 6.0, [952] := 6.0, [953] := 6.0, [954] := 6.0, [955] := 6.0, [956] := 6.0, [957] := 6.0, [958] := 6.0, [959] := 6.0,
        [960] := 6.0, [961] := 6.0, [962] := 6.0, [963] := 6.0, [964] := 6.0, [965] := 6.0, [966] := 6.0, [967] := 6.0, [968] := 6.0, [969] := 6.0, [970] := 6.0, [971] := 6.0, [972] := 6.0, [973] := 6.0, [974] := 6.0, [975] := 6.0, [976] := 6.0, [977] := 6.0, [978] := 6.0, [979] := 6.0, [980] := 6.0, [981] := 6.0, [982] := 6.0, [983] := 6.0, [984] := 6.0, [985] := 6.0, [986] := 6.0, [987] := 6.0, [988] := 6.0, [989] := 6.0, [990] := 6.0, [991] := 6.0, [992] := 6.0, [993] := 6.0, [994] := 6.0, [995] := 6.0, [996] := 6.0, [997] := 6.0, [998] := 6.0, [999] := 6.0);
   p29r18_winder_b_selected_diam_inch : REAL := 6.0;   // Winder Winder B Diameter Calculation Selected Diameter [in]
   p29r18_winder_b_unload : REAL := 3.25;
   p29r20 : routine := (comment := -1073738505, warning := 2, warning_ack := 2, state := 3);   // Winder Winder Turret VFD
        .FAULT.0   // Winder Liner Winder VFD Drive Fault
        .FAULT.2   // Winder Winder Turret VFD Drive Not Ready
        .FAULT.3   // Winder Winder Turret VFD Drive Not in Remote Mode
        .FAULT.4   // Winder Winder Turret VFD Motor Temperature Fault
        .WARNING.0   // Winder Winder Turret VFD Drive Warning
        .WARNING.1   // Winder Winder Turret VFD No Winder Selected
        .UNACK_FAULT   // Winder Winder Turret VFD Unacknowleged Faults Exist
        .UNACK_WARNING   // Winder Winder Turret VFD Unacknowleged Warnings Exist
        .STATE.0   // Winder Winder Turret One Step Per Scan
        .STATE.1   // Winder Winder Turret Step 1: Idle
        .STATE.2   // Winder Turret Step 2: Start Index Direction
        .STATE.3   // Winder Winder Turret Step 3: Index Active
        .STATE.4   // Winder Winder Turret Step 4: Prox Positive Transition
        .STATE.5   // Winder Winder Turret Step 5: Drive Stop
        .STATE.6   // Winder Winder Turret Step 6: Index Complete
        .STATE.7   // Winder Winder Turret Step 7:Stop Drive
        .STATE.8   // Winder Winder Turret Step 8: Index Complete
   p29r20_acc_dec_ramp : SYS_ACC_DEC_RAMP := (IN_param_master_accel_rate := 2.0, IN_param_master_decel_rate := 2.0, IN_last_scan_s := 0.032558);   // Winder Winder Turret VFD Accel / Decel Ramp
   p29r20_accel_rate : REAL := 2.0;   // Winder Winder Turret VFD Accel Rate
   p29r20_decel_rate : REAL := 2.0;   // Winder Winder Turret VFD Decel Rate
   p29r20_fast_accel : REAL := 2.0;
   p29r20_fast_decel : REAL := 2.0;
   p29r20_index_complete : BOOL := 1;   // Winder Winder Turret VFD Index Complete
   p29r20_index_move_timer : TIMER;   // Winder Winder Turret VFD Move Timer
   p29r20_permissive : BOOL := 1;   // Winder Winder Turret VFD Permissive
   p29r20_request_fwd : BOOL;   // Winder Winder Turret VFD Request Index FWD
   p29r20_request_rev : BOOL;   // Winder Winder Turret VFD Request Index REV
   p29r20_selected_speed : REAL;   // Winder Winder Turret VFD Selected Speed
   p29r20_timer_fault : TIMER[10];   // Winder Winder Turret VFD Fault Dwell Timer
   p29r20_timer_warning : TIMER[4] := ([1].ACC := 33, [1].EN := 1, [1].DN := 1);   // Winder Winder Turret VFD Warning Dwell Timer
   p29r20_zero_speed : BOOL := 1;   // Winder Winder Turret Zero Speed
   p30_di_pin_1 : BOOL := 1;   // Retraction System Inputs Pin 1 Stowed
   p30_di_pin_2 : BOOL := 1;   // Retraction System Inputs Pin 2 Stowed
   p30_di_pin_3 : BOOL := 1;   // Retraction System Inputs Pin 3 Stowed
   p30_di_pin_4 : BOOL := 1;   // Retraction System Inputs Pin 4 Stowed
   p30_di_pin_5 : BOOL := 1;   // Retraction System Inputs Pin 5 Stowed
   p30_di_pin_6 : BOOL := 1;   // Retraction System Inputs Pin 6 Stowed
   p30_di_pin_7 : BOOL := 1;   // Retraction System Inputs Pin 7 Stowed
   p30_di_pin_8 : BOOL := 1;   // Retraction System Inputs Pin 8 Stowed
   p30_di_retraction_down_ls : BOOL := 1;   // Retraction System Digital Input LS: Down
   p30_di_retraction_up_ls : BOOL;   // Retraction System Digital Input Operator Side LS: Up
   p30_di_rotation_fault : BOOL;   // Retraction System Digital Input Rotation Fault
   p30_di_ss_close : BOOL;   // Retraction System Digital Input SS: Open/Off/Close Close
   p30_di_ss_open : BOOL;   // Retraction System Digital Input SS: Open/Off/Close Open
   p30_dint_to_hmi : DINT[16] := ([0] := 255);   // Retraction System Dint to HMI
        [0].0   // Retraction System Dint to HMI Safety Pin 1 Stowed
        [0].1   // Retraction System Dint to HMI Safety Pin 2 Stowed
        [0].2   // Retraction System Dint to HMI Safety Pin 3 Stowed
        [0].3   // Retraction System Dint to HMI Safety Pin 4 Stowed
        [0].4   // Retraction System Dint to HMI Safety Pin 5 Stowed
        [0].5   // Retraction System Dint to HMI Safety Pin 6 Stowed
        [0].6   // Retraction System Dint to HMI Safety Pin 7 Stowed
        [0].7   // Retraction System Dint to HMI Safety Pin 8 Stowed
        [2].0   // Retraction System Alarms A00: Rotation Fault
        [2].1   // Retraction System Alarms A01:
        [2].2   // Retraction System Alarms A02:
        [2].3   // Retraction System Alarms A03:
        [2].4   // Retraction System Alarms A04:
        [2].5   // Retraction System Alarms A05:
        [2].6   // Retraction System Alarms A06:
        [2].7   // Retraction System Alarms A07:
        [2].8   // Retraction System Alarms A08:
        [2].9   // Retraction System Alarms A09
        [2].10   // Retraction System Alarms A10:
        [2].11   // Retraction System Alarms A11:
        [2].12   // Retraction System Alarms A12:
        [2].13   // Retraction System Alarms A13:
        [2].14   // Retraction System Alarms A14:
        [2].15   // Retraction System Alarms A15:
        [2].16   // Retraction System Alarms A16:
        [2].17   // Retraction System Alarms A17:
        [2].18   // Retraction System Alarms A18:
        [2].19   // Retraction System Alarms A19:
        [2].20   // Retraction System Alarms A20:
        [2].21   // Retraction System Alarms A21:
        [2].22   // Retraction System Alarms A22:
        [2].23   // Retraction System Alarms A23:
        [2].24   // Retraction System Alarms A24:
        [2].25   // Retraction System Alarms A25:
        [2].26   // Retraction System Alarms A26:
        [2].27   // Retraction System Alarms A27:
        [2].28   // Retraction System Alarms A28:
        [2].29   // Retraction System Alarms A29:
        [2].30   // Retraction System Alarms A30:
        [2].31   // Retraction System Alarms A31:
        [4].0   // Retraction System Warnings W00:
        [4].1   // Retraction System Warnings W01:
        [4].2   // Retraction System Warnings W02:
        [4].3   // Retraction System Warnings W03:
        [4].4   // Retraction System Warnings W04:
        [4].5   // Retraction System Warnings W05:
        [4].6   // Retraction System Warnings W06:
        [4].7   // Retraction System Warnings W07:
        [4].8   // Retraction System Warnings W08:
        [4].9   // Retraction System Warnings W09
        [4].10   // Retraction System Warnings W10:
        [4].11   // Retraction System Warnings W11:
        [4].12   // Retraction System Warnings W12:
        [4].13   // Retraction System Warnings W13:
        [4].14   // Retraction System Warnings W14:
        [4].15   // Retraction System Warnings W15:
        [4].16   // Retraction System Warnings W16:
        [4].17   // Retraction System Warnings W17:
        [4].18   // Retraction System Warnings W18:
        [4].19   // Retraction System Warnings W19:
        [4].20   // Retraction System Warnings W20:
        [4].21   // Retraction System Warnings W21:
        [4].22   // Retraction System Warnings W22:
        [4].23   // Retraction System Warnings W23:
        [4].24   // Retraction System Warnings W24:
        [4].25   // Retraction System Warnings W25:
        [4].26   // Retraction System Warnings W26:
        [4].27   // Retraction System Warnings W27:
        [4].28   // Retraction System Warnings W28:
        [4].29   // Retraction System Warnings W29:
        [4].30   // Retraction System Warnings W30:
        [4].31   // Retraction System Warnings W31:
   p30_do_retract_motion : BOOL;
   p30_do_retract_reset : BOOL;
   p30_do_rotation_fwd : BOOL;   // Retraction System Output Retraction FWD
   p30_do_rotation_rev : BOOL;   // Retraction System Output Retraction REV
   p30_real_to_hmi : REAL[112];   // Retraction System Real to HMI
   p30r01 : routine := (comment := 7);   // Retraction System
   p30r02 : routine := (comment := -1073741761);   // Retraction System Misc Control
   p30r02_fault_exists : BOOL;
   p30r02_timer_fault : TIMER[4];   // Retraction System Misc Control Fault Dwell Timer
   p30r02_timer_warning : TIMER[4];   // Retraction System Misc Control Warning Dwell Timer
   p30r02_unack_fault : BOOL;   // Retraction System Misc Control Unacknoledged Fault Exist
   p30r02_unack_warning : BOOL;   // Retraction System Misc Control Unacknoledge Warning Exist
   p30r02_warning_exists : BOOL;
   p30r03 : routine := (comment := -1073741761);   // Retraction System Input
   p30r03_timer_fault : TIMER[4];   // Retraction System Input Fault Dwell Timer
   p30r03_timer_warning : TIMER[4];   // Retraction System Input Warning Dwell Timer
   p30r04 : routine := (comment := -1073741761);   // Retraction System Output
   p30r04_timer_fault : TIMER[4];   // Retraction System Output Fault Dwell Timer
   p30r04_timer_warning : TIMER[4];   // Retraction System Output Warning Dwell Timer
   p30r05 : routine := (comment := -1073741761);   // Retraction System Dint to HMI
   p30r05_timer_fault : TIMER[4];   // Retraction System Dint to HMI Fault Dwell Timer
   p30r05_timer_warning : TIMER[4];   // Retraction System Dint to HMI Warning Dwell Timer
   p30r06 : routine := (comment := -1073741572);   // Retraction System Real to HMI
   p30r06_timer_fault : TIMER[4];   // Retraction System Real to HMI Fault Dwell Timer
   p30r06_timer_warning : TIMER[4];   // Retraction System Real to HMI Warning Dwell Timer
   p30r07 : routine := (comment := -1073741761);   // Retraction System Alarms
   p30r07_timer_fault : TIMER[4];   // Retraction System Alarms Fault Dwell Timer
   p30r07_timer_warning : TIMER[4];   // Retraction System Alarms Warning Dwell Timer
   p30r08 : routine := (comment := -1073741761);   // Retraction System Warnings
   p30r08_timer_fault : TIMER[4];   // Retraction System Warnings Fault Dwell Timer
   p30r08_timer_warning : TIMER[4];   // Retraction System Warnings Warning Dwell Timer
   p30r09 : routine := (comment := -1073741761);   // Retraction System Modes
   p30r09_mode_close : BOOL;   // Retraction System Modes Close Mode
   p30r09_mode_off : BOOL := 1;   // Retraction System Modes Off Mode
   p30r09_mode_open : BOOL;   // Retraction System Modes Open Mode
   p30r09_timer_fault : TIMER[4];   // Retraction System Modes Fault Dwell Timer
   p30r09_timer_warning : TIMER[4];   // Retraction System Modes Warning Dwell Timer
   p30r10 : routine := (comment := -1073741777);   // Retraction System Retraction
        .FAULT.0   // Retraction System Retraction Rotation Fault
        .WARNING.0   // Retraction System Retraction Pins Not Stowed
   p30r10_motion_monitor_dwell : TIMER := (PRE := 500);
   p30r10_request_close : BOOL;   // Retraction System Retraction Request Close
   p30r10_request_monitor : BOOL;
   p30r10_request_open : BOOL;   // Retraction System Retraction Request Open
   p30r10_run_permissive : BOOL := 1;   // Retraction System Retraction Run Permissive
   p30r10_safety_pins_stowed : BOOL := 1;   // Retraction System Retraction All Safety Pins Stowed
   p30r10_state : DINT;   // Splice Press Sequence State
        .0   // Splice Press Sequence State 0 One Step Per Scan
        .1   // Splice Press Sequence State 1 Idle
        .2   // Splice Press Sequence State 2 Enable Sequence
        .3   // Splice Press Sequence State 3 Close Exit Clamp
        .4   // Splice Press Sequence State 4 Close Inlet Clamp
        .5   // Splice Press Sequence State 5 Closing Platen
        .6   // Splice Press Sequence State 6 Cure in Progress
        .7   // Splice Press Sequence State 7 Cure Done
        .8   // Splice Press Sequence State 8 Platen Open
        .9   // Splice Press Sequence State 9 Inlet Clamp Open
        .10   // Splice Press Sequence State 10 Exit Clamp Open
        .11   // Splice Press Sequence State 11 Complete
   p30r10_timer_fault : TIMER[4] := ([1].PRE := 400);   // Retraction System Retraction Fault Dwell Timer
   p30r10_timer_warning : TIMER[4] := ([0].PRE := 1000);   // Retraction System Retraction Warning Dwell Timer
   p31r09 : routine;   // Edge Control Modes
        .UNACK_FAULT   // Edge Control Modes Unacknowledged Fault Exists
        .UNACK_WARNING   // Edge Control Modes Unacknowledged Warning Exists
   p32r13_request_auto_stop : BOOL;   // Impreg Supply VFD Request Auto Stop
   retraction_delay_timer : TIMER := (PRE := 4000);
   retraction_delay_timer_2 : TIMER := (PRE := 4000);
   spring_spd_adj_prcnt : REAL := 0.975;
   turret_in_position : BOOL := 1;   // Turret In Position
   winder_ramped_setpoint : REAL;
END_VAR

PROGRAM P01_Main   (* main routine R01_Main *)
VAR
   PIDE_02 : PID_ENHANCED := (PV := 60.0, PVEUMax := 500.0, SPOper := 60.0, SPHLimit := 200.0, RatioProg := 1.0, RatioOper := 1.0, RatioHLimit := 1.0, RatioLLimit := 1.0, CVProg := 50.0, CVOper := 50.0, CVEUMax := 100.0, CVHLimit := 100.0, PGain := 5.0, IGain := 0.1, PVEDerivative := 1, DSmoothing := 1, PVTracking := 1, PVHHLimit := 1000.0, PVHLimit := 900.0, PVLLimit := -1000.0, PVLLLimit := -2000.0, DevHHLimit := 1000.0, DevHLimit := 1000.0, ManualAfterInit := 1, ProgManualReq := 1, RTSTime := 1, CVEU := 50.0, CV := 50.0, SP := 60.0, SPPercent := 12.0, PVPercent := 12.0, InitPrimary := 1, Ratio := 1.0, DevLAlarm := 1, DevLLAlarm := 1, ProgOper := 1, Manual := 1, DeltaT := 0.1, AtuneBusy := 1);
END_VAR

ROUTINE R01_Main   (* ladder *)
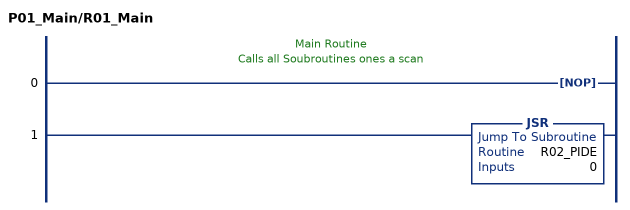
   // Main Routine
   // Calls all Soubroutines ones a scan
   0: NOP();
   1: JSR(R02_PIDE,0);
END_ROUTINE

ROUTINE R02_PIDE   (* function block diagram *)
   SHEET 1
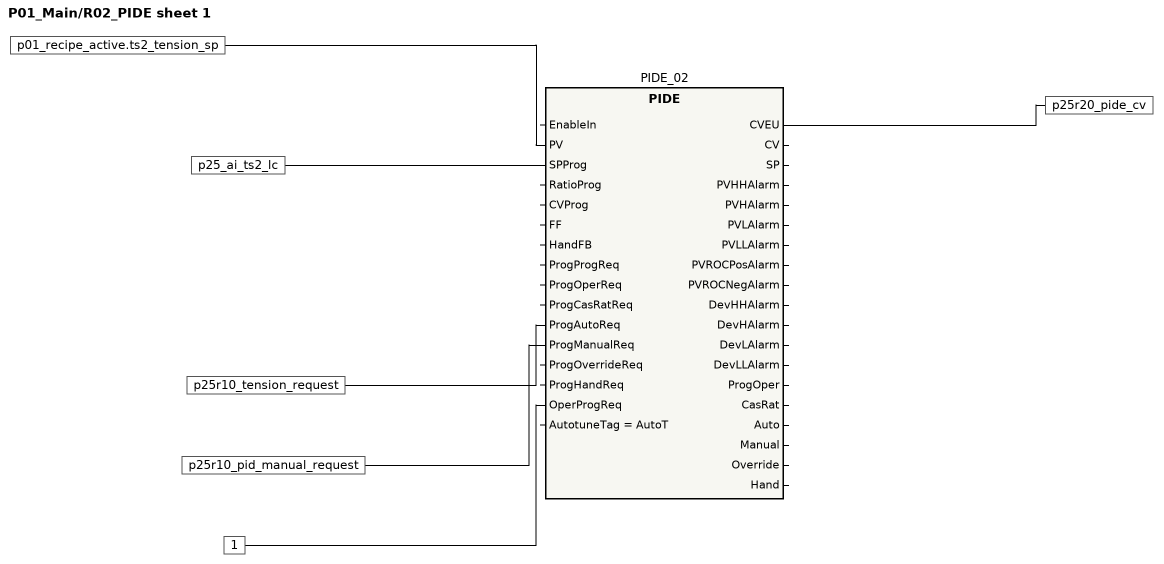
   PIDE_02 : PIDE(PV := p01_recipe_active.ts2_tension_sp, SPProg := p25_ai_ts2_lc, ProgAutoReq := p25r10_tension_request, ProgManualReq := p25r10_pid_manual_request, OperProgReq := 1, AutotuneTag := AutoT);   // unwired pins: EnableIn RatioProg CVProg FF HandFB ProgProgReq ProgOperReq ProgCasRatReq ProgOverrideReq ProgHandReq CV SP PVHHAlarm PVHAlarm PVLAlarm PVLLAlarm PVROCPosAlarm PVROCNegAlarm DevHHAlarm DevHAlarm DevLAlarm DevLLAlarm ProgOper CasRat Auto Manual Override Hand
   p25r20_pide_cv := PIDE_02.CVEU;
END_ROUTINE
END_PROGRAM

PROGRAM P01_System   (* main routine R01_Main *)
VAR
   Limit_Clamp : sys_Limit_Clamp;   // Limit Clamp
   tmrFlash : TIMER[4] := ([0].PRE := 1000, [0].ACC := 1000, [0].EN := 1, [0].DN := 1, [1].PRE := 1000, [1].ACC := 1005, [1].EN := 1, [1].DN := 1, [2].PRE := 500, [2].EN := 1, [2].TT := 1, [3].PRE := 500);   // Flash Timer
END_VAR

ROUTINE R01_Main   (* ladder *)
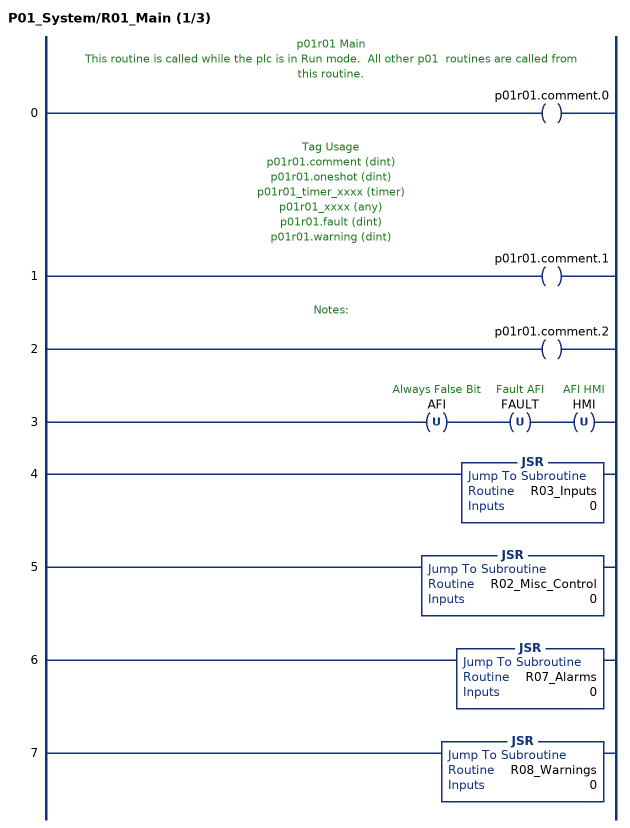
   // p01r01 Main
   // This routine is called while the plc is in Run mode.  All other p01  routines are called from this routine.
   0: OTE(p01r01.comment.0);
   // Tag Usage
   // p01r01.comment (dint)
   // p01r01.oneshot (dint)
   // p01r01_timer_xxxx (timer)
   // p01r01_xxxx (any)
   // p01r01.fault (dint)
   // p01r01.warning (dint)
   1: OTE(p01r01.comment.1);
   // Notes:
   2: OTE(p01r01.comment.2);
   3: OTU(AFI)OTU(FAULT)OTU(HMI);
   4: JSR(R03_Inputs,0);
   5: JSR(R02_Misc_Control,0);
   6: JSR(R07_Alarms,0);
   7: JSR(R08_Warnings,0);
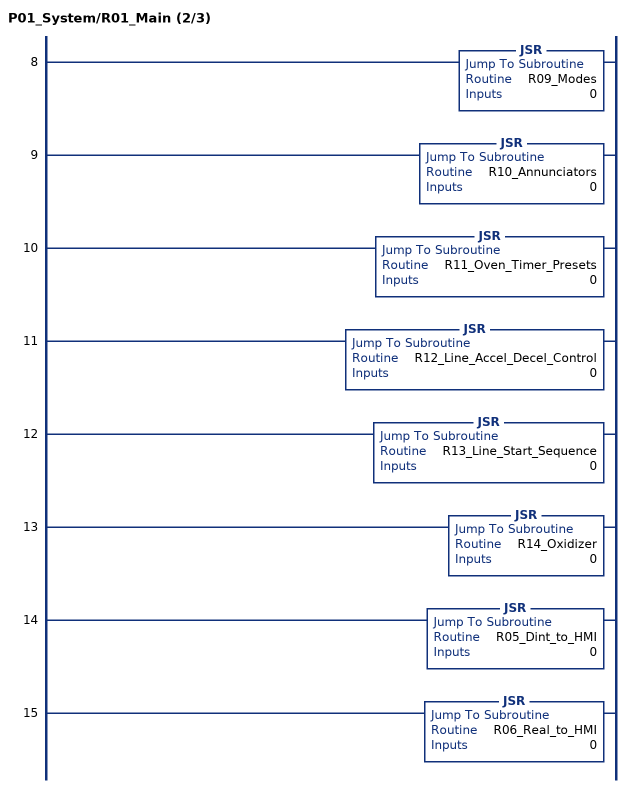
   8: JSR(R09_Modes,0);
   9: JSR(R10_Annunciators,0);
   10: JSR(R11_Oven_Timer_Presets,0);
   11: JSR(R12_Line_Accel_Decel_Control,0);
   12: JSR(R13_Line_Start_Sequence,0);
   13: JSR(R14_Oxidizer,0);
   14: JSR(R05_Dint_to_HMI,0);
   15: JSR(R06_Real_to_HMI,0);
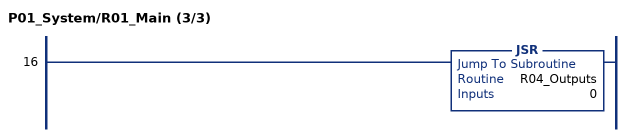
   16: JSR(R04_Outputs,0);
END_ROUTINE

ROUTINE R02_Misc_Control   (* ladder *)
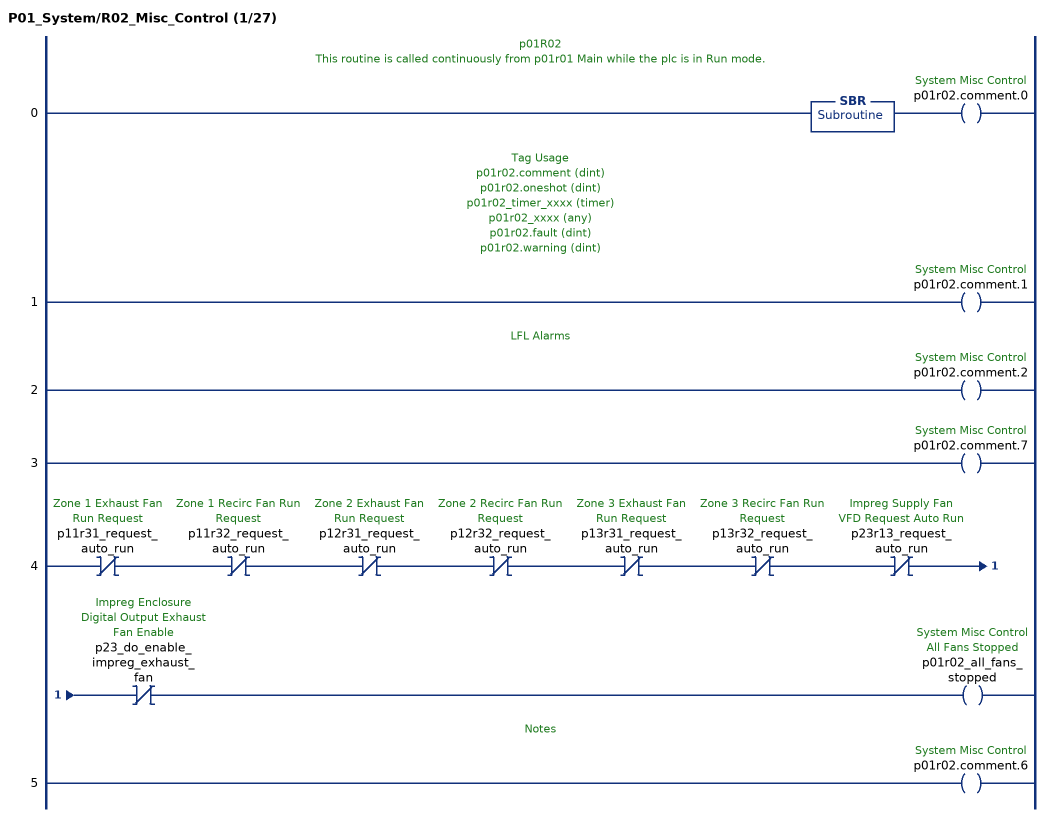
   // p01R02
   // This routine is called continuously from p01r01 Main while the plc is in Run mode.
   0: SBR()OTE(p01r02.comment.0);
   // Tag Usage
   // p01r02.comment (dint)
   // p01r02.oneshot (dint)
   // p01r02_timer_xxxx (timer)
   // p01r02_xxxx (any)
   // p01r02.fault (dint)
   // p01r02.warning (dint)
   1: OTE(p01r02.comment.1);
   // LFL Alarms
   2: OTE(p01r02.comment.2);
   3: OTE(p01r02.comment.7);
   4: XIO(p11r31_request_auto_run)XIO(p11r32_request_auto_run)XIO(p12r31_request_auto_run)XIO(p12r32_request_auto_run)XIO(p13r31_request_auto_run)XIO(p13r32_request_auto_run)XIO(p23r13_request_auto_run)XIO(p23_do_enable_impreg_exhaust_fan)OTE(p01r02_all_fans_stopped);
   // Notes
   5: OTE(p01r02.comment.6);
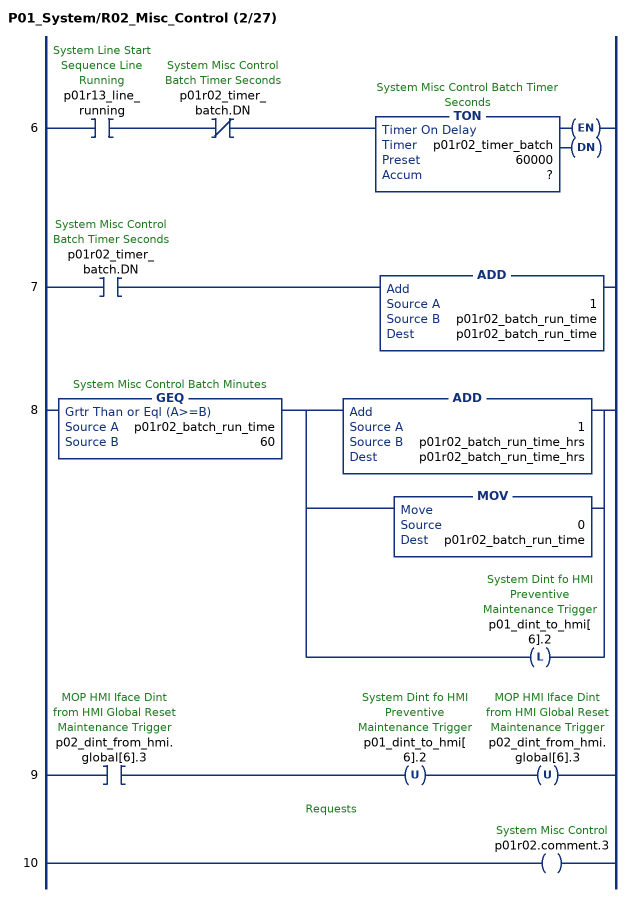
   6: XIC(p01r13_line_running)XIO(p01r02_timer_batch.DN)TON(p01r02_timer_batch,?,?);
   7: XIC(p01r02_timer_batch.DN)ADD(1,p01r02_batch_run_time,p01r02_batch_run_time);
   8: GEQ(p01r02_batch_run_time,60)[ADD(1,p01r02_batch_run_time_hrs,p01r02_batch_run_time_hrs) ,MOV(0,p01r02_batch_run_time) ,OTL(p01_dint_to_hmi[6].2) ];
   9: XIC(p02_dint_from_hmi.global[6].3)OTU(p01_dint_to_hmi[6].2)OTU(p02_dint_from_hmi.global[6].3);
   // Requests
   10: OTE(p01r02.comment.3);
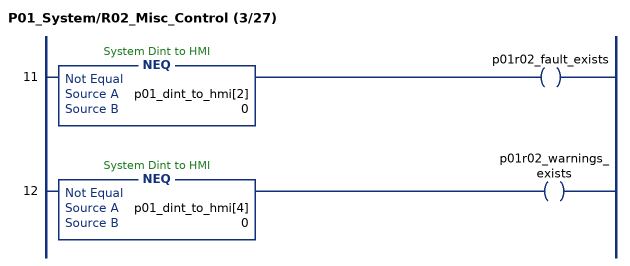
   11: NEQ(p01_dint_to_hmi[2],0)OTE(p01r02_fault_exists);
   12: NEQ(p01_dint_to_hmi[4],0)OTE(p01r02_warnings_exists);
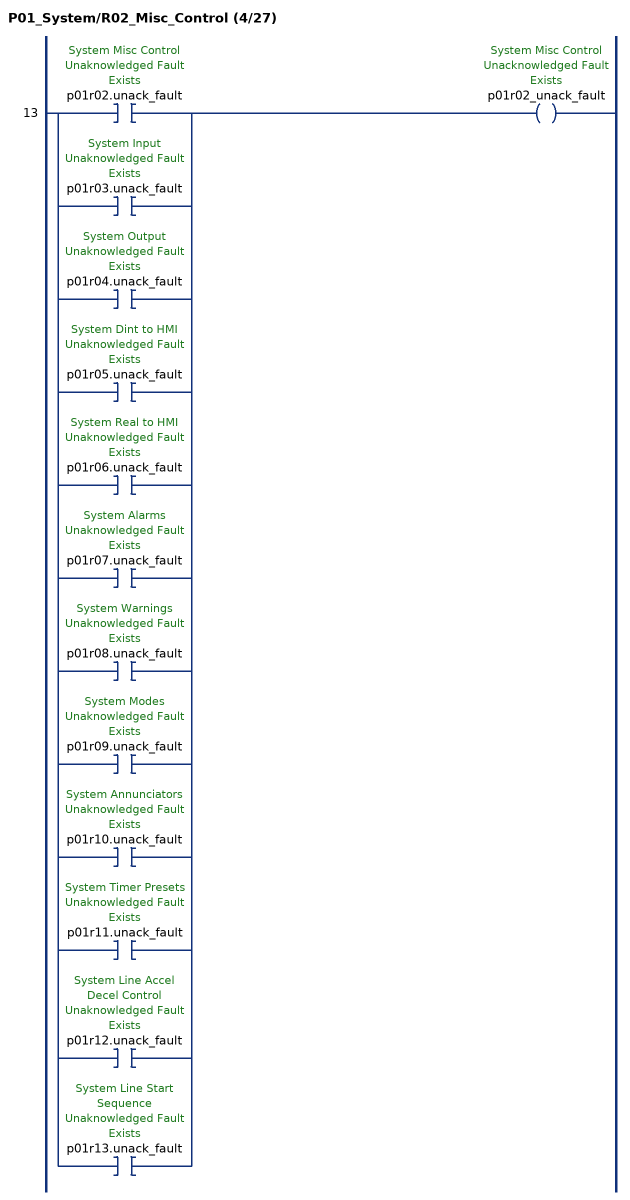
   13: [XIC(p01r02.unack_fault) ,XIC(p01r03.unack_fault) ,XIC(p01r04.unack_fault) ,XIC(p01r05.unack_fault) ,XIC(p01r06.unack_fault) ,XIC(p01r07.unack_fault) ,XIC(p01r08.unack_fault) ,XIC(p01r09.unack_fault) ,XIC(p01r10.unack_fault) ,XIC(p01r11.unack_fault) ,XIC(p01r12.unack_fault) ,XIC(p01r13.unack_fault) ]OTE(p01r02_unack_fault);
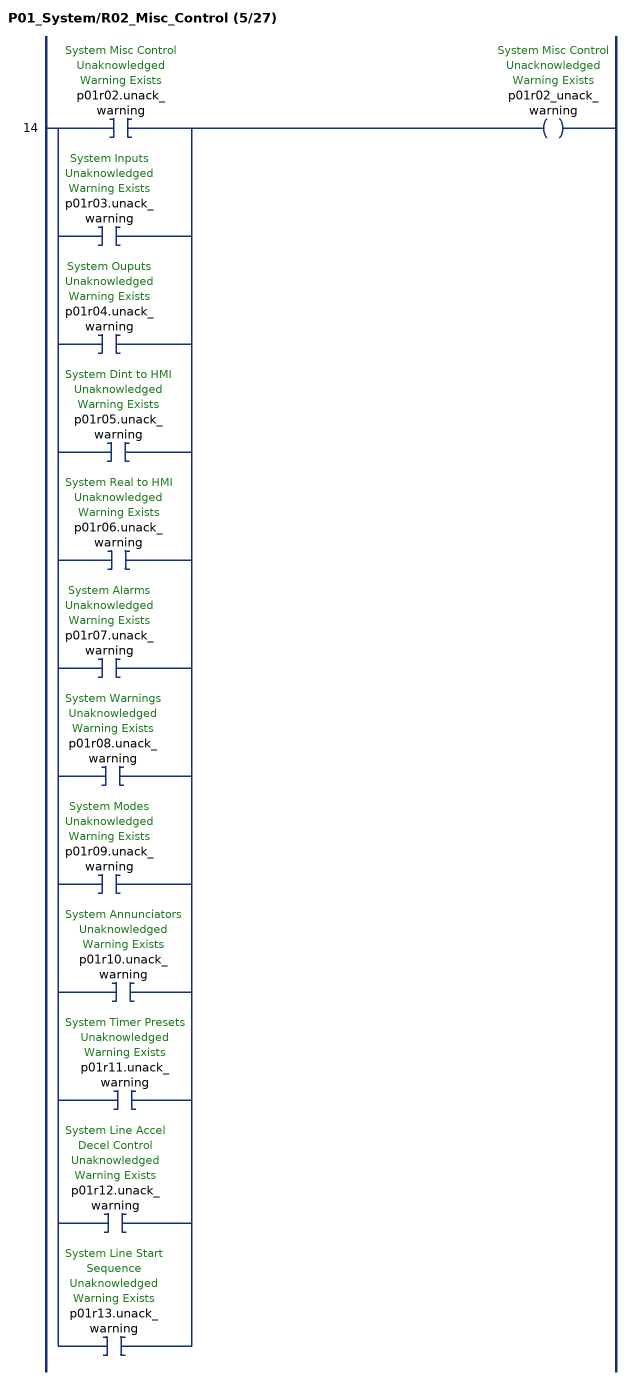
   14: [XIC(p01r02.unack_warning) ,XIC(p01r03.unack_warning) ,XIC(p01r04.unack_warning) ,XIC(p01r05.unack_warning) ,XIC(p01r06.unack_warning) ,XIC(p01r07.unack_warning) ,XIC(p01r08.unack_warning) ,XIC(p01r09.unack_warning) ,XIC(p01r10.unack_warning) ,XIC(p01r11.unack_warning) ,XIC(p01r12.unack_warning) ,XIC(p01r13.unack_warning) ]OTE(p01r02_unack_warning);
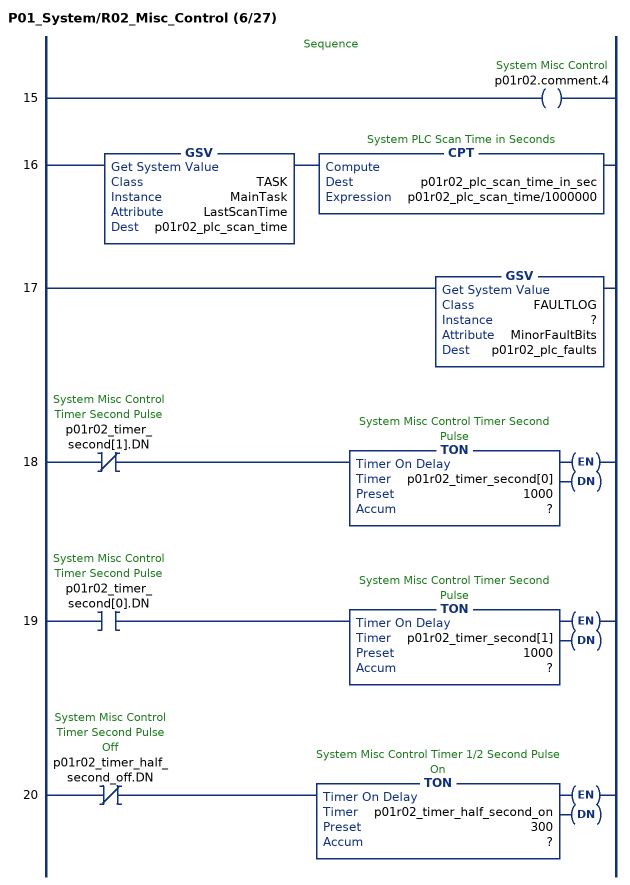
   // Sequence
   15: OTE(p01r02.comment.4);
   16: GSV(TASK,MainTask,LastScanTime,p01r02_plc_scan_time)CPT(p01r02_plc_scan_time_in_sec,p01r02_plc_scan_time/1000000);
   17: GSV(FAULTLOG,?,MinorFaultBits,p01r02_plc_faults);
   18: XIO(p01r02_timer_second[1].DN)TON(p01r02_timer_second[0],?,?);
   19: XIC(p01r02_timer_second[0].DN)TON(p01r02_timer_second[1],?,?);
   20: XIO(p01r02_timer_half_second_off.DN)TON(p01r02_timer_half_second_on,?,?);
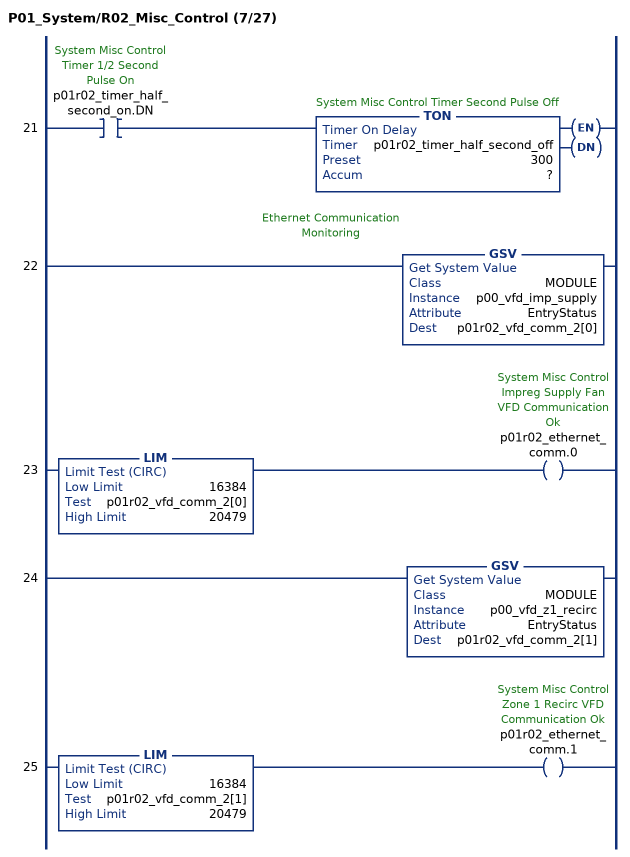
   21: XIC(p01r02_timer_half_second_on.DN)TON(p01r02_timer_half_second_off,?,?);
   // Ethernet Communication
   // Monitoring
   22: GSV(MODULE,p00_vfd_imp_supply,EntryStatus,p01r02_vfd_comm_2[0]);
   23: LIM(16384,p01r02_vfd_comm_2[0],20479)OTE(p01r02_ethernet_comm.0);
   24: GSV(MODULE,p00_vfd_z1_recirc,EntryStatus,p01r02_vfd_comm_2[1]);
   25: LIM(16384,p01r02_vfd_comm_2[1],20479)OTE(p01r02_ethernet_comm.1);
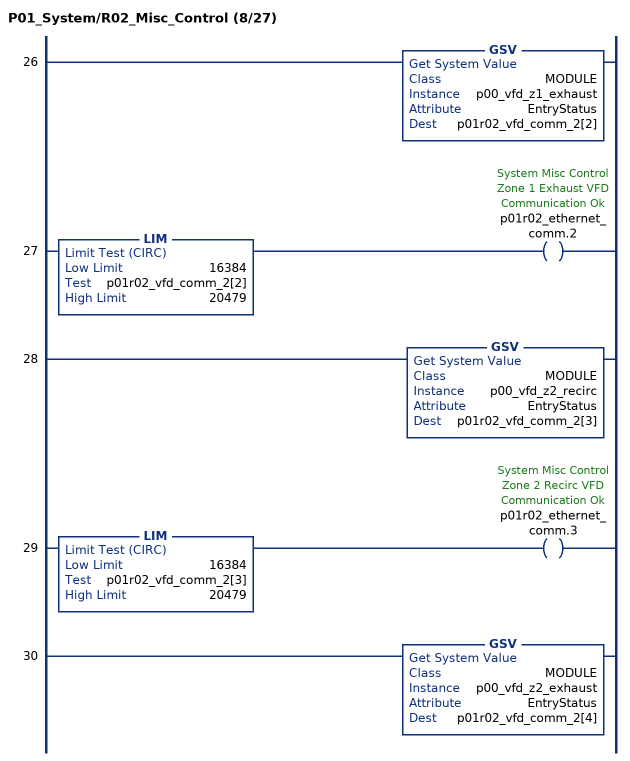
   26: GSV(MODULE,p00_vfd_z1_exhaust,EntryStatus,p01r02_vfd_comm_2[2]);
   27: LIM(16384,p01r02_vfd_comm_2[2],20479)OTE(p01r02_ethernet_comm.2);
   28: GSV(MODULE,p00_vfd_z2_recirc,EntryStatus,p01r02_vfd_comm_2[3]);
   29: LIM(16384,p01r02_vfd_comm_2[3],20479)OTE(p01r02_ethernet_comm.3);
   30: GSV(MODULE,p00_vfd_z2_exhaust,EntryStatus,p01r02_vfd_comm_2[4]);
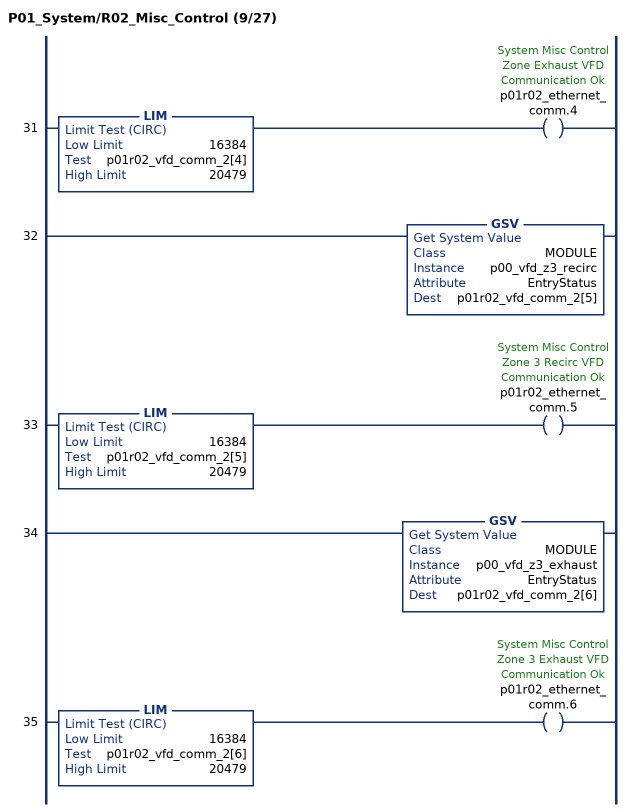
   31: LIM(16384,p01r02_vfd_comm_2[4],20479)OTE(p01r02_ethernet_comm.4);
   32: GSV(MODULE,p00_vfd_z3_recirc,EntryStatus,p01r02_vfd_comm_2[5]);
   33: LIM(16384,p01r02_vfd_comm_2[5],20479)OTE(p01r02_ethernet_comm.5);
   34: GSV(MODULE,p00_vfd_z3_exhaust,EntryStatus,p01r02_vfd_comm_2[6]);
   35: LIM(16384,p01r02_vfd_comm_2[6],20479)OTE(p01r02_ethernet_comm.6);
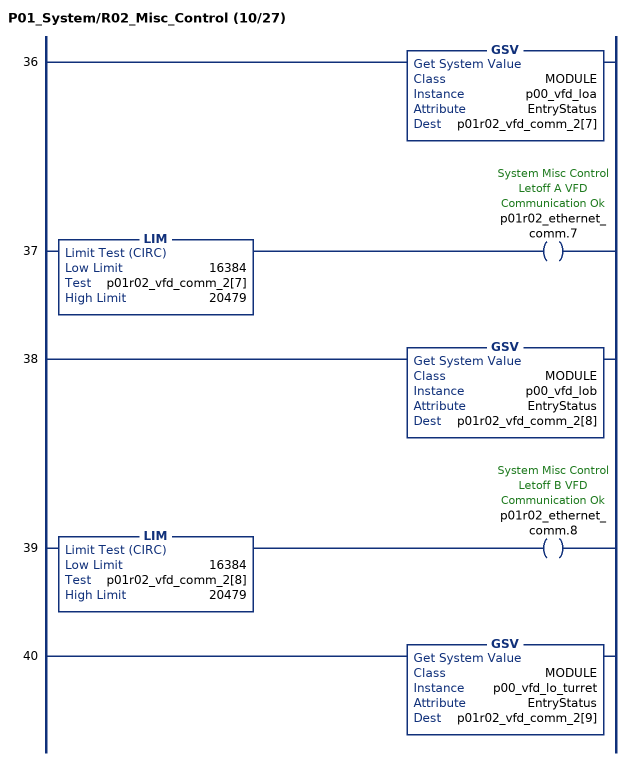
   36: GSV(MODULE,p00_vfd_loa,EntryStatus,p01r02_vfd_comm_2[7]);
   37: LIM(16384,p01r02_vfd_comm_2[7],20479)OTE(p01r02_ethernet_comm.7);
   38: GSV(MODULE,p00_vfd_lob,EntryStatus,p01r02_vfd_comm_2[8]);
   39: LIM(16384,p01r02_vfd_comm_2[8],20479)OTE(p01r02_ethernet_comm.8);
   40: GSV(MODULE,p00_vfd_lo_turret,EntryStatus,p01r02_vfd_comm_2[9]);
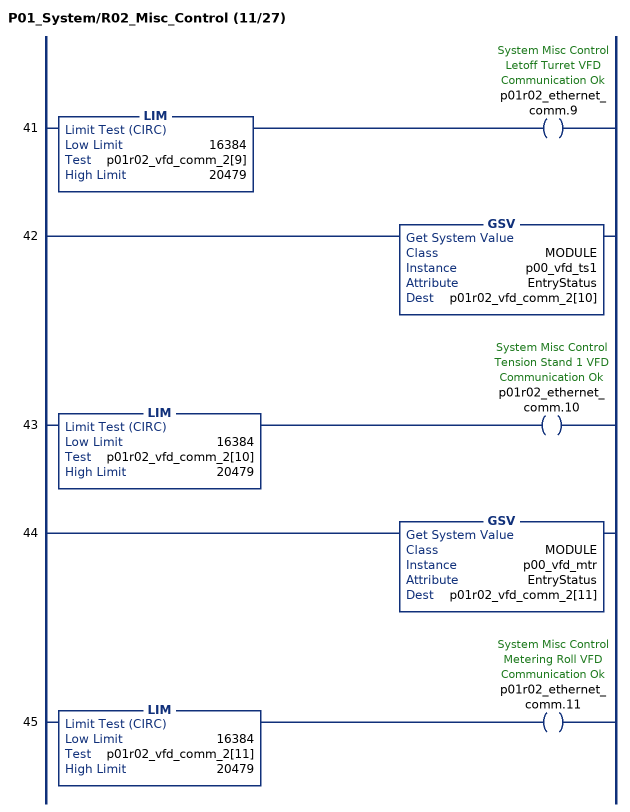
   41: LIM(16384,p01r02_vfd_comm_2[9],20479)OTE(p01r02_ethernet_comm.9);
   42: GSV(MODULE,p00_vfd_ts1,EntryStatus,p01r02_vfd_comm_2[10]);
   43: LIM(16384,p01r02_vfd_comm_2[10],20479)OTE(p01r02_ethernet_comm.10);
   44: GSV(MODULE,p00_vfd_mtr,EntryStatus,p01r02_vfd_comm_2[11]);
   45: LIM(16384,p01r02_vfd_comm_2[11],20479)OTE(p01r02_ethernet_comm.11);
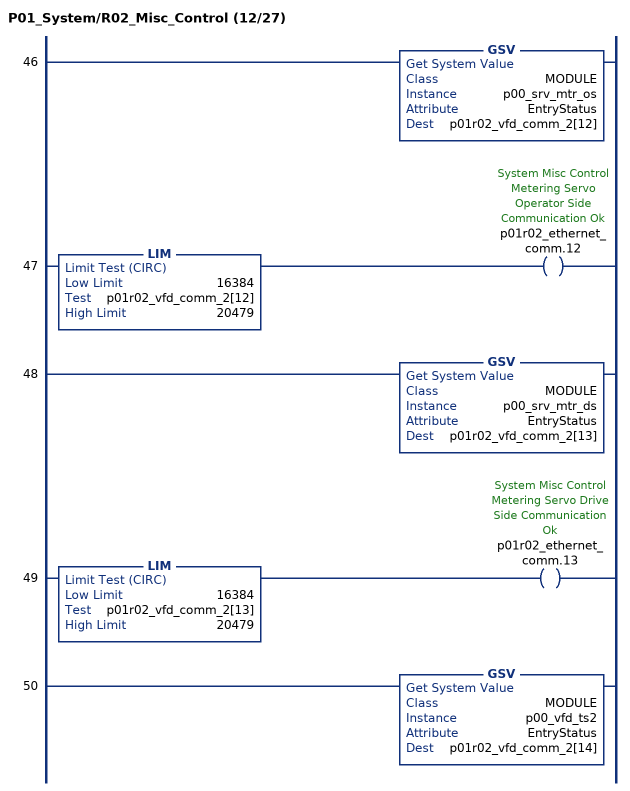
   46: GSV(MODULE,p00_srv_mtr_os,EntryStatus,p01r02_vfd_comm_2[12]);
   47: LIM(16384,p01r02_vfd_comm_2[12],20479)OTE(p01r02_ethernet_comm.12);
   48: GSV(MODULE,p00_srv_mtr_ds,EntryStatus,p01r02_vfd_comm_2[13]);
   49: LIM(16384,p01r02_vfd_comm_2[13],20479)OTE(p01r02_ethernet_comm.13);
   50: GSV(MODULE,p00_vfd_ts2,EntryStatus,p01r02_vfd_comm_2[14]);
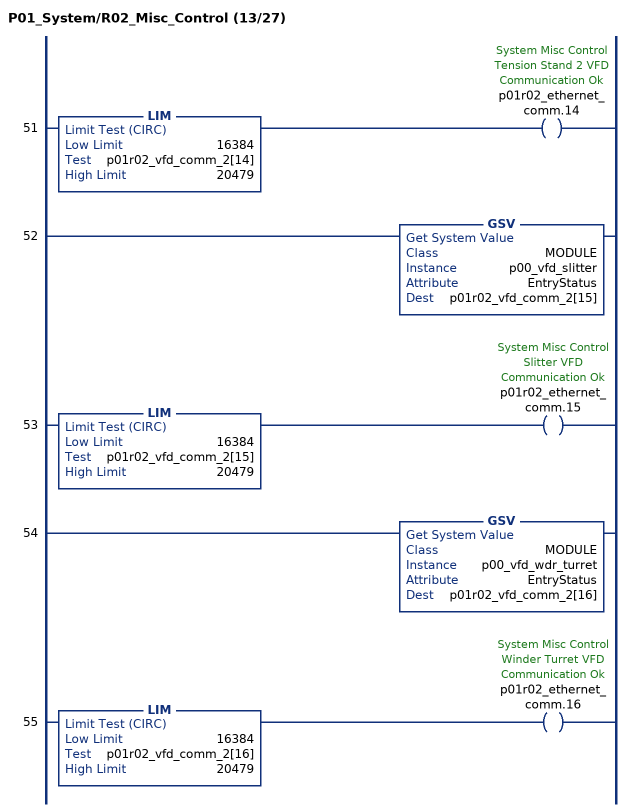
   51: LIM(16384,p01r02_vfd_comm_2[14],20479)OTE(p01r02_ethernet_comm.14);
   52: GSV(MODULE,p00_vfd_slitter,EntryStatus,p01r02_vfd_comm_2[15]);
   53: LIM(16384,p01r02_vfd_comm_2[15],20479)OTE(p01r02_ethernet_comm.15);
   54: GSV(MODULE,p00_vfd_wdr_turret,EntryStatus,p01r02_vfd_comm_2[16]);
   55: LIM(16384,p01r02_vfd_comm_2[16],20479)OTE(p01r02_ethernet_comm.16);
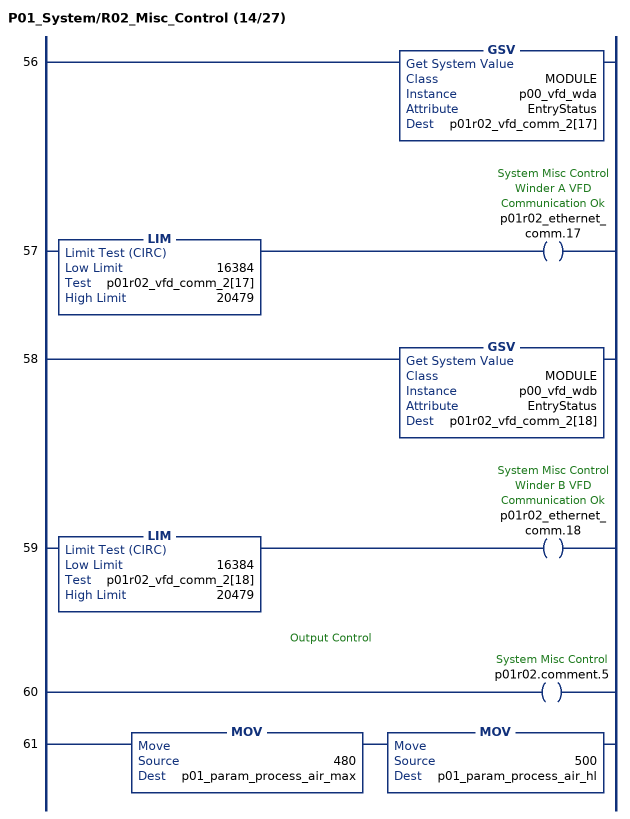
   56: GSV(MODULE,p00_vfd_wda,EntryStatus,p01r02_vfd_comm_2[17]);
   57: LIM(16384,p01r02_vfd_comm_2[17],20479)OTE(p01r02_ethernet_comm.17);
   58: GSV(MODULE,p00_vfd_wdb,EntryStatus,p01r02_vfd_comm_2[18]);
   59: LIM(16384,p01r02_vfd_comm_2[18],20479)OTE(p01r02_ethernet_comm.18);
   // Output Control
   60: OTE(p01r02.comment.5);
   61: MOV(480,p01_param_process_air_max)MOV(500,p01_param_process_air_hl);
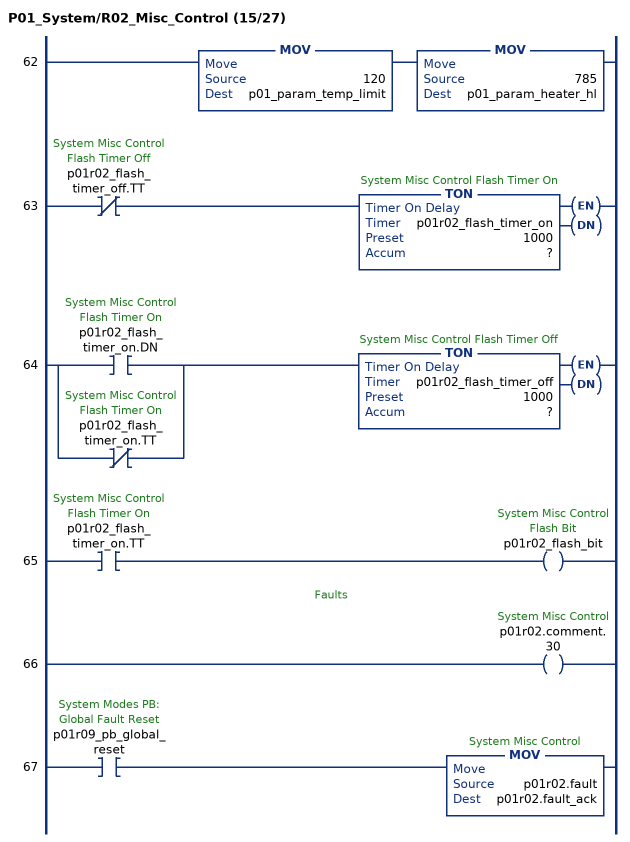
   62: MOV(120,p01_param_temp_limit)MOV(785,p01_param_heater_hl);
   63: XIO(p01r02_flash_timer_off.TT)TON(p01r02_flash_timer_on,?,?);
   64: [XIC(p01r02_flash_timer_on.DN) ,XIO(p01r02_flash_timer_on.TT) ]TON(p01r02_flash_timer_off,?,?);
   65: XIC(p01r02_flash_timer_on.TT)OTE(p01r02_flash_bit);
   // Faults
   66: OTE(p01r02.comment.30);
   67: XIC(p01r09_pb_global_reset)MOV(p01r02.fault,p01r02.fault_ack);
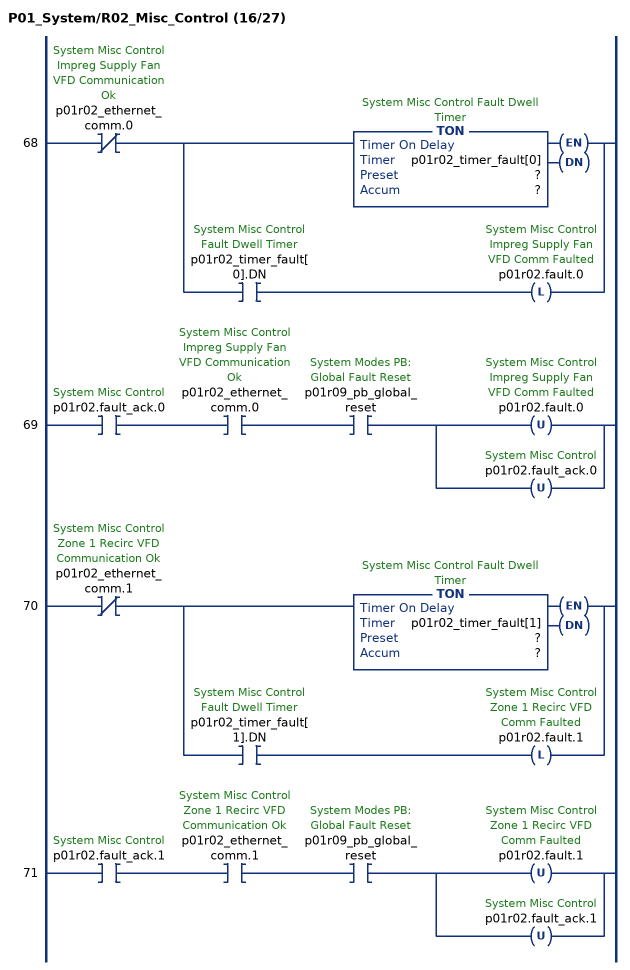
   68: XIO(p01r02_ethernet_comm.0)[TON(p01r02_timer_fault[0],?,?) ,XIC(p01r02_timer_fault[0].DN) OTL(p01r02.fault.0) ];
   69: XIC(p01r02.fault_ack.0)XIC(p01r02_ethernet_comm.0)XIC(p01r09_pb_global_reset)[OTU(p01r02.fault.0) ,OTU(p01r02.fault_ack.0) ];
   70: XIO(p01r02_ethernet_comm.1)[TON(p01r02_timer_fault[1],?,?) ,XIC(p01r02_timer_fault[1].DN) OTL(p01r02.fault.1) ];
   71: XIC(p01r02.fault_ack.1)XIC(p01r02_ethernet_comm.1)XIC(p01r09_pb_global_reset)[OTU(p01r02.fault.1) ,OTU(p01r02.fault_ack.1) ];
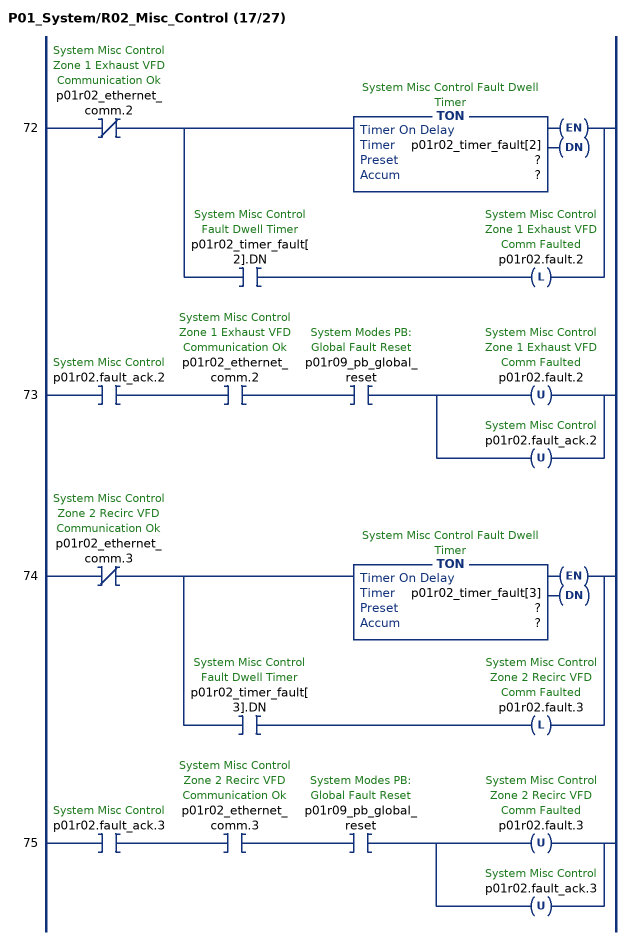
   72: XIO(p01r02_ethernet_comm.2)[TON(p01r02_timer_fault[2],?,?) ,XIC(p01r02_timer_fault[2].DN) OTL(p01r02.fault.2) ];
   73: XIC(p01r02.fault_ack.2)XIC(p01r02_ethernet_comm.2)XIC(p01r09_pb_global_reset)[OTU(p01r02.fault.2) ,OTU(p01r02.fault_ack.2) ];
   74: XIO(p01r02_ethernet_comm.3)[TON(p01r02_timer_fault[3],?,?) ,XIC(p01r02_timer_fault[3].DN) OTL(p01r02.fault.3) ];
   75: XIC(p01r02.fault_ack.3)XIC(p01r02_ethernet_comm.3)XIC(p01r09_pb_global_reset)[OTU(p01r02.fault.3) ,OTU(p01r02.fault_ack.3) ];
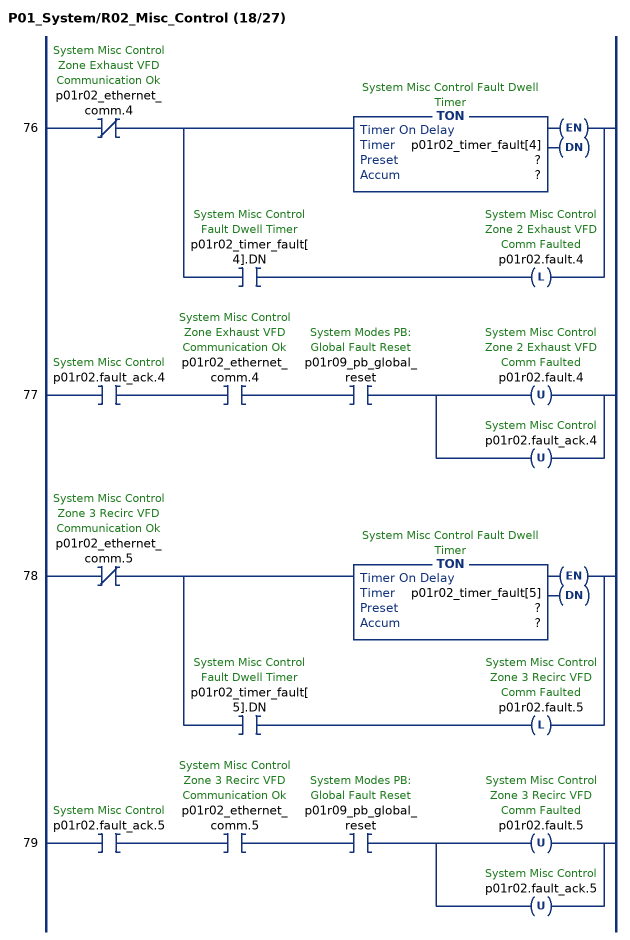
   76: XIO(p01r02_ethernet_comm.4)[TON(p01r02_timer_fault[4],?,?) ,XIC(p01r02_timer_fault[4].DN) OTL(p01r02.fault.4) ];
   77: XIC(p01r02.fault_ack.4)XIC(p01r02_ethernet_comm.4)XIC(p01r09_pb_global_reset)[OTU(p01r02.fault.4) ,OTU(p01r02.fault_ack.4) ];
   78: XIO(p01r02_ethernet_comm.5)[TON(p01r02_timer_fault[5],?,?) ,XIC(p01r02_timer_fault[5].DN) OTL(p01r02.fault.5) ];
   79: XIC(p01r02.fault_ack.5)XIC(p01r02_ethernet_comm.5)XIC(p01r09_pb_global_reset)[OTU(p01r02.fault.5) ,OTU(p01r02.fault_ack.5) ];
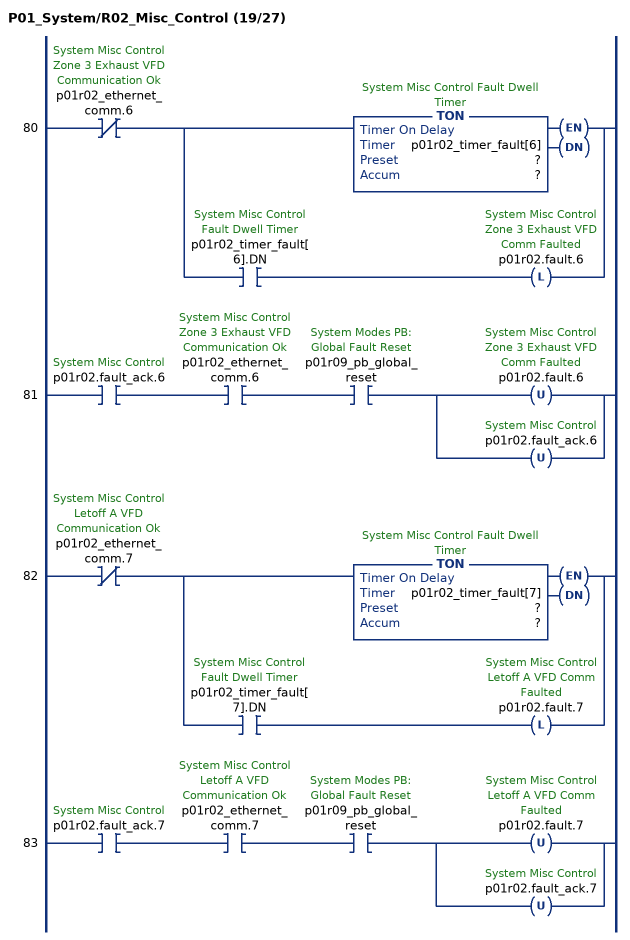
   80: XIO(p01r02_ethernet_comm.6)[TON(p01r02_timer_fault[6],?,?) ,XIC(p01r02_timer_fault[6].DN) OTL(p01r02.fault.6) ];
   81: XIC(p01r02.fault_ack.6)XIC(p01r02_ethernet_comm.6)XIC(p01r09_pb_global_reset)[OTU(p01r02.fault.6) ,OTU(p01r02.fault_ack.6) ];
   82: XIO(p01r02_ethernet_comm.7)[TON(p01r02_timer_fault[7],?,?) ,XIC(p01r02_timer_fault[7].DN) OTL(p01r02.fault.7) ];
   83: XIC(p01r02.fault_ack.7)XIC(p01r02_ethernet_comm.7)XIC(p01r09_pb_global_reset)[OTU(p01r02.fault.7) ,OTU(p01r02.fault_ack.7) ];
